IF eError <> MotionlinxAI_Error_States.NO_ERROR  OR eError = MotionlinxAI_Error_States.MOTOR_UNDERVOLTAGE  THEN
	IF (bMotorDisconnected AND NOT bMotorExpected)  THEN
		_Error := FALSE;
	ELSE
		_Error := TRUE;
		eError := eError;
	
			
//		IF oClearMotorError = 0 THEN
//			oClearMotorError := 1;
//		ELSIF oClearMotorError = 1 THEN
//			oClearMotorError := 0;
//		END_IF;
	END_IF

ELSE
	_Error := FALSE;
END_IF;
END_ACTION

PROPERTY HasFault : BOOL
GET
HasFault := eMotionlinxAIState < MotionlinxAI_States.HOMING;// or bCommunicationsFailed;
END_GET
END_PROPERTY

METHOD PROTECTED HMICommunication
VAR_INPUT
END_VAR
SUPER^.HMICommunication();

//Handle the requests to extend and retract
IF ComponentBase_HMI.Status.HMIControlAvailable THEN
	IF MotionlinxAI_HMI.Command.Extend THEN
//		Extend();
	ELSIF MotionlinxAI_HMI.Command.Retract THEN
//		Retract();
	END_IF
END_IF

//Update HMI status info
//Cylinder_HMI.Status.Extended	:= _Extended;
//Cylinder_HMI.Status.Extending	:= _Extending;
//Cylinder_HMI.Status.Retracted	:= _Retracted;
//Cylinder_HMI.Status.Retracting	:= _Retracting;
//Cylinder_HMI.Config.ExtendTime	:= _ExtendTime;
//Cylinder_HMI.Config.RetractTime := _RetractTime;
END_METHOD

//! @summary Basic component initialization logic
METHOD PROTECTED Initialize : BOOL;

//! @description This method is called by <c>CyclicLogic()</c> as required



//Set the cylinder to retracted
//oMotorAccel	:= 500;		//From recipe value here
//IF Output THEN
//	_Extended  := TRUE;
//	_Retracted := FALSE;
//ELSE
//	_Extended  := FALSE;
//	_Retracted := TRUE;
//END_IF



//Call base class Initialize
Initialize := SUPER^.Initialize();
END_METHOD

PROPERTY IsReady : BOOL
GET
IsReady := eMotionlinxAIState > MotionlinxAI_States.HOMING;
END_GET
END_PROPERTY

PROPERTY MaxSpeed : uint
SET
uMaxSpeed	:= MaxSpeed;
END_SET
END_PROPERTY

METHOD PROTECTED Monitoring
VAR_INPUT
END_VAR
_Busy	 := NOT Stopped;//MotionlinxAI_Motor_Status:=3 OR MotionlinxAI_Motor_Status:=4 ;
_Error	 := eError>0 OR eMotionlinxAIState < MotionlinxAI_States.HOMING;;
_ErrorID := eError;
SUPER^.Monitoring();
END_METHOD

PROPERTY MotorDisconnected : bool
GET
MotorDisconnected	:= bMotorDisconnected;
END_GET
END_PROPERTY

METHOD RaiseAlarm2Args
VAR_IN_OUT
	Alarm : FB_TcAlarm; //Alarm to be raised
END_VAR

VAR_INPUT
	String_1 : STRING; //First String Parameter (The Name of this component will be applied first automatically)
	String_2 : STRING; //Second String Parameter
END_VAR
F_RaiseAlarmWithStringParameters(Alarm	  := Alarm,
								 String_1 := Name,
								 String_2 := String_1,
								 String_3 := String_2);
END_METHOD

METHOD Start : BOOL
VAR_INPUT
END_VAR
IF bEnabled THEN 
	oMotorControl.0 := TRUE;
	oMotorBrakeMode  := 2;
END_IF
END_METHOD

METHOD Stop
VAR_INPUT
END_VAR
oMotorControl.0 := FALSE;
oMotorBrakeMode := 2;
END_METHOD

PROPERTY Stopped : bool
GET
Stopped	:= bAxis_Stopped;
END_GET
END_PROPERTY

PROPERTY Velocity : int
SET
nRequestedSpeed	:= Velocity;
//Recipe.Axis.Acceleration := Acceleration;
END_SET
END_PROPERTY

END_FUNCTION_BLOCK

// ---- Machine/Components/MotionLinxAI/Controller/FB_MotionlinxAI_Controller.TcPOU
(*	
*)
FUNCTION_BLOCK FB_MotionlinxAI_Controller EXTENDS FB_ComponentBase IMPLEMENTS I_MotionlinxAI_Controller_Sts
VAR
//Inputs
	iSensors AT%I* : INT;
	iSysDiagnostics AT%I* : BYTE;
//	Drive_1_Left	  : FB_MotionlinxAI_Axis (Main_Sensor	:= iSensors.4, Aux_Sensor	:= iSensors.0 ):= (Name := 'Left Drive 1');
//	Drive_2_Right	  : FB_MotionlinxAI_Axis (Main_Sensor	:= iSensors.6, Aux_Sensor	:= iSensors.2 ):= (Name := 'Right Drive 2');
	

	//Output
	oServoControl AT%Q* : INT;
	oSetPin2Out AT%Q* : BYTE;
	oClearMotorError  AT%Q* : BYTE;
	
	//From Other project, can possibly be modifdied a bit
	//Connection Monitoring//
	bWCState AT%I* : BOOL; //0 is Data Valid, 1 is Data Invalid
	
	tonCommunicationsFailed : TON;
	bCommunicationsFailed : BOOL;
	
	bInputToggle AT%I* : BOOL;

	// Internal variables
	//Error Resetting//
	bError : BOOL;
	tpErrorReset : TP;
	
	//Speed Limits//
	rPGDMaxSpeed : REAL := 536.0;
	rPGDMinSpeed : REAL := 3888.0;
	
	
	//Motor Status//
	eMotorStatus: MotionlinxAI_Motor_Status;
	eErrorRecord : MotionlinxAI_Error_States;
	_stController_Sts	:ST_Controller_Status;

	
	
	
//	_ExtendRequest	: BOOL;
//	_RetractRequest : BOOL;
//	_Extended		: BOOL;
//	_Retracted		: BOOL;
//	_Extending		: BOOL;
//	_Retracting		: BOOL;
//	_ExtendTime		: LREAL := 1000; // Default time 1s
//	_RetractTime	: LREAL := 1000; // Default time 1s

//	// Timer for Extend/Retract
//	Extend_TON	  : TON;
//	Retract_TON	  : TON;
//	Extend_RTRIG  : R_TRIG;
//	Retract_RTRIG : R_TRIG;

	//HMI 
	MotionlinxAI_Controller_HMI : ST_MotionlinxAI_Axis_HMI;
END_VAR

PROPERTY CommunicationsFailed : bool
GET
CommunicationsFailed	:= bCommunicationsFailed;
END_GET
END_PROPERTY

PROPERTY Controller_Status : ST_Controller_Status
GET
Controller_Status	:= _stController_Sts;
END_GET
END_PROPERTY

METHOD PROTECTED CreateEvents
VAR_INPUT
END_VAR
SUPER^.CreateEvents();
END_METHOD

METHOD CyclicLogic
VAR

END_VAR
//////////Error Handling//////////
errorCheck();
_stController_Sts.Sensors	:= iSensors;
_stController_Sts.bEnabled	:= isEnabled;
_stController_Sts.HasFault	:= HasFault;

//////////Set Speed Limits//////////
//uLMinSpeed := 15+uLMaxSpeed/100;
//uRMinSpeed := 15+uRMaxSpeed/100;
//////////Set Speeds//////////
//oMotorLSpeed := LIMIT(UINT_TO_INT(uLMinSpeed),UINT_TO_INT(nRequestedSpeedLeft),UINT_TO_INT(uLMaxSpeed));
//oMotorRSpeed := LIMIT(UINT_TO_INT(uRMinSpeed),UINT_TO_INT(nRequestedSpeedRight),UINT_TO_INT(uRMaxSpeed));


////////////Stop On Disable//////////
//IF NOT bEnabled THEN
//	oMotorLDecel := oMotorRDecel := 500;	
//	oMotorLControl.0 := oMotorRControl.0 := FALSE;
//ELSE
//	oMotorLDecel := oMotorRDecel := 500;
//END_IF;



//////////Communications Monitoring//////////
tonCommunicationsFailed(IN:= bWCState, PT:= T#10S, Q => bCommunicationsFailed);


//One shot the requests


//Handle Extend
//IF Extend_RTRIG.Q THEN
//	Output			:= TRUE;
//	_Extending		:= TRUE;
//	_Retracting		:= FALSE;
//	_Retracted		:= FALSE;
//	_RetractRequest := FALSE;
//END_IF

//Handle Retract
//IF Retract_RTRIG.Q THEN
//	Output		   := FALSE;
//	_Extending	   := FALSE;
//	_Retracting	   := TRUE;
//	_Extended	   := FALSE;
//	_ExtendRequest := FALSE;
//END_IF

//Handle the time to Extend/Retract
//Extend_TON(IN := _Extending, PT := LREAL_TO_TIME(_ExtendTime));
//Retract_TON(IN := _Retracting, PT := LREAL_TO_TIME(_RetractTime));
//IF Extend_TON.Q THEN
//	_Extended  := TRUE;
//	_Extending := FALSE;
//END_IF

//IF Retract_TON.Q THEN
//	_Retracted	:= TRUE;
//	_Retracting := FALSE;
//END_IF

SUPER^.CyclicLogic();
END_METHOD

METHOD Disable : BOOL
(*BRAKING MODES:
	0 : NORMAL - HOLDS IN PLACE BY SHORTING WINDINGS
	1 : FREE - NOT HELD IN PLACE
	2 : SERVO - MAINTAINS POSITION BASED ON HALLS EFFECT SENSOR*)
//oMotorLDecel := oMotorRDecel := 500;
//bEnabled := FALSE;
//(*oMotorLControl.0 := FALSE;
//oMotorRControl.0 := FALSE;*)
//oMotorLBrakeMode := oMotorRBrakeMode := 2;
END_METHOD

METHOD EmergencyStop : BOOL
(*BRAKING MODES:
	0 : NORMAL - HOLDS IN PLACE BY SHORTING WINDINGS
	1 : FREE - NOT HELD IN PLACE
	2 : SERVO - MAINTAINS POSITION BASED ON HALLS EFFECT SENSOR*)
//oMotorLDecel := oMotorRDecel := 1;
//bEnabled := FALSE;
//(*oMotorLControl.0 := FALSE;
//oMotorRControl.0 := FALSE;*)
//oMotorLBrakeMode := oMotorRBrakeMode := 0;
END_METHOD

METHOD Enable : BOOL
(*BRAKING MODES:
	0 : NORMAL - HOLDS IN PLACE BY SHORTING WINDINGS
	1 : FREE - NOT HELD IN PLACE
	2 : SERVO - MAINTAINS POSITION BASED ON HALLS EFFECT SENSOR*)
//bEnabled := TRUE;
//oMotorLBrakeMode := oMotorRBrakeMode := 2;
END_METHOD

ACTION errorCheck:
//oClearMotorError := 0;




//IF eErrorLeft <> MotionlinxAI_Error_States.NO_ERROR OR eErrorRight <> MotionlinxAI_Error_States.NO_ERROR OR eErrorLeft = MotionlinxAI_Error_States.MOTOR_UNDERVOLTAGE OR eErrorRight = MotionlinxAI_Error_States.MOTOR_UNDERVOLTAGE THEN
//	IF (bLeftMotorDisconnected AND NOT bLeftMotorExpected) OR (bRightMotorDisconnected AND NOT bRightMotorExpected) THEN
//		bError := FALSE;
//	ELSE
//		bError := TRUE;
//	//	eErrorRecordLeft := eErrorLeft;
//	//	eErrorRecordRight := eErrorRight;
			
//		IF oClearMotorError = 0 THEN
//			oClearMotorError := 1;
//		ELSIF oClearMotorError = 1 THEN
//			oClearMotorError := 0;
//		END_IF;
//	END_IF

//ELSE
//	bError := FALSE;
//END_IF;
END_ACTION

PROPERTY FaultLocation : STRING(50)
GET
//FaultLocation := sDriveName;
END_GET
END_PROPERTY

PROPERTY HasFault : BOOL
GET
//HasFault := eMotionlinxAIState < MotionlinxAI_States.HOMING or bCommunicationsFailed;
END_GET
END_PROPERTY

METHOD PROTECTED HMICommunication
VAR_INPUT
END_VAR
SUPER^.HMICommunication();

//Handle the requests to extend and retract
IF ComponentBase_HMI.Status.HMIControlAvailable THEN
	IF MotionlinxAI_Controller_HMI.Command.Extend THEN
	//	Extend();
	ELSIF MotionlinxAI_Controller_HMI.Command.Retract THEN
	//	Retract();
	END_IF
END_IF

//Update HMI status info
//MotionlinxAI_Controller_HMI.Status.Extended	:= _Extended;
//MotionlinxAI_Controller_HMI.Status.Extending	:= _Extending;
//MotionlinxAI_Controller_HMI.Status.Retracted	:= _Retracted;
//MotionlinxAI_Controller_HMI.Status.Retracting	:= _Retracting;
//MotionlinxAI_Controller_HMI.Config.ExtendTime	:= _ExtendTime;
//MotionlinxAI_Controller_HMI.Config.RetractTime := _RetractTime;
END_METHOD

//! @summary Basic component initialization logic
METHOD PROTECTED Initialize : BOOL;

//! @description This method is called by <c>CyclicLogic()</c> as required
//Set the cylinder to retracted
//IF Output THEN
//	_Extended  := TRUE;
//	_Retracted := FALSE;
//ELSE
//	_Extended  := FALSE;
//	_Retracted := TRUE;
//END_IF

//_Extending		:= FALSE;
//_ExtendRequest	:= FALSE;
//_Retracting		:= FALSE;
//_RetractRequest := FALSE;

//Call base class Initialize
Initialize := SUPER^.Initialize();
END_METHOD

PROPERTY IsEnabled : BOOL
GET
//IsEnabled := bEnabled;
END_GET
END_PROPERTY

PROPERTY IsReady : BOOL
GET
//IsReady := eMotionlinxAIState > MotionlinxAI_States.HOMING;
END_GET
END_PROPERTY

METHOD PROTECTED Monitoring
VAR_INPUT
END_VAR
//_Busy	 := _Extending OR _Retracting;
_Error	 := bCommunicationsFailed;
_ErrorID := 0;
SUPER^.Monitoring();
END_METHOD

PROPERTY Sensors : int
GET
Sensors	:= iSensors;
END_GET
END_PROPERTY

ACTION stop:
//oMotorLControl.0 := FALSE;
//oMotorRControl.0 := FALSE;
END_ACTION

END_FUNCTION_BLOCK

// ---- Machine/Components/Robots/UR/fbUR.TcPOU
FUNCTION_BLOCK fbUR
VAR_INPUT
END_VAR
VAR_OUTPUT
END_VAR
VAR	
	EIO_UR_Outputs AT %Q* : UR_Output_Data;
	EIO_UR_Inputs  AT %I* : UR_Safety_Bits_Data;

	bBrakeRelease AT %Q* : BOOL;
	
	rtRobotSafe			: R_TRIG;
	
	tpBrakeRelease		: TP;
	
	tonPowerUpRobot		: TON;
	tpPowerOnPulse		: TP;
END_VAR

rtRobotSafe(CLK := EIO_UR_Inputs.data.ibNormalMode OR EIO_UR_Inputs.data.ibReducedMode);
EIO_UR_Outputs.data.obBrakeRelease := bBrakeRelease;

tpBrakeRelease(IN := GVL_Safety.PALLETISER_ESTOP_OK AND NOT (GVL_HMI.ibResetButton OR GVL_HMI.bHMIResetButton), PT := T#1S, Q => bBrakeRelease);

tonPowerUpRobot(IN:= NOT GVL_Palletiser.ibURPowered, PT := T#20S);
tpPowerOnPulse(IN := tonPowerUpRobot.Q, Q => GVL_Palletiser.obURPowerOn, PT := T#0.5S);

END_FUNCTION_BLOCK

// ---- Machine/Components/Contactor/FB_Contactor.TcPOU
(*	This FB is used for a single output solenoid 
	It uses the times to say when Extended/Retracted  	
	It starts assuming retracted and the output off.
*)
FUNCTION_BLOCK FB_Contactor EXTENDS FB_ComponentBase IMPLEMENTS I_Contactor
VAR
    //Output
    Output AT %Q* : BOOL;

    // Internal variables
    _ExtendRequest  : BOOL;
    _RetractRequest : BOOL;
    _Extended       : BOOL;
    _Retracted      : BOOL;
    _Extending      : BOOL;
    _Retracting     : BOOL;
    _ExtendTime     : LREAL := 1000; // Default time 1s
    _RetractTime    : LREAL := 1000; // Default time 1s

    // Timer for Extend/Retract
    Extend_TON    : TON;
    Retract_TON   : TON;
    Extend_RTRIG  : R_TRIG;
    Retract_RTRIG : R_TRIG;

    //HMI 
    Contactor_HMI : ST_Contactor_HMI;
END_VAR

METHOD PROTECTED CreateEvents
VAR_INPUT
END_VAR
SUPER^.CreateEvents();
END_METHOD

METHOD CyclicLogic
//One shot the requests
Extend_RTRIG(CLK := _ExtendRequest);
Retract_RTRIG(CLK := _RetractRequest);

//Handle Extend
IF Extend_RTRIG.Q THEN
    Output          := TRUE;
    _Extending      := TRUE;
    _Retracting     := FALSE;
    _Retracted      := FALSE;
    _RetractRequest := FALSE;
END_IF

//Handle Retract
IF Retract_RTRIG.Q THEN
    Output         := FALSE;
    _Extending     := FALSE;
    _Retracting    := TRUE;
    _Extended      := FALSE;
    _ExtendRequest := FALSE;
END_IF

//Handle the time to Extend/Retract
Extend_TON(IN := _Extending, PT := LREAL_TO_TIME(_ExtendTime));
Retract_TON(IN := _Retracting, PT := LREAL_TO_TIME(_RetractTime));
IF Extend_TON.Q THEN
    _Extended  := TRUE;
    _Extending := FALSE;
END_IF

IF Retract_TON.Q THEN
    _Retracted  := TRUE;
    _Retracting := FALSE;
END_IF

SUPER^.CyclicLogic();
END_METHOD

METHOD Extend
_ExtendRequest  := TRUE;
_RetractRequest := FALSE;
END_METHOD

PROPERTY Extended : BOOL
GET
Extended := _Extended;
END_GET
END_PROPERTY

PROPERTY ExtendTime : LREAL
GET
ExtendTime := _ExtendTime;
END_GET
SET
END_SET
END_PROPERTY

METHOD PROTECTED HMICommunication
VAR_INPUT
END_VAR
SUPER^.HMICommunication();

//Handle the requests to extend and retract
IF ComponentBase_HMI.Status.HMIControlAvailable THEN
    IF Contactor_HMI.Command.Extend THEN
        Extend();
    ELSIF Contactor_HMI.Command.Retract THEN
        Retract();
    END_IF
END_IF

//Update HMI status info
Contactor_HMI.Status.Extended    := _Extended;
Contactor_HMI.Status.Extending   := _Extending;
Contactor_HMI.Status.Retracted   := _Retracted;
Contactor_HMI.Status.Retracting  := _Retracting;
Contactor_HMI.Config.ExtendTime  := _ExtendTime;
Contactor_HMI.Config.RetractTime := _RetractTime;
END_METHOD

//! @summary Basic component initialization logic
METHOD PROTECTED Initialize : BOOL;

//! @description This method is called by <c>CyclicLogic()</c> as required
//Set the Contactor to retracted
IF Output THEN
    _Extended  := TRUE;
    _Retracted := FALSE;
ELSE
    _Extended  := FALSE;
    _Retracted := TRUE;
END_IF

_Extending      := FALSE;
_ExtendRequest  := FALSE;
_Retracting     := FALSE;
_RetractRequest := FALSE;

//Call base class Initialize
Initialize := SUPER^.Initialize();
END_METHOD

METHOD PROTECTED Monitoring
VAR_INPUT
END_VAR
_Busy    := _Extending OR _Retracting;
_Error   := FALSE;
_ErrorID := 0;
SUPER^.Monitoring();
END_METHOD

METHOD Retract
_ExtendRequest  := FALSE;
_RetractRequest := TRUE;
END_METHOD

PROPERTY Retracted : BOOL
GET
Retracted := _Retracted;
END_GET
END_PROPERTY

PROPERTY RetractTime : LREAL
GET
RetractTime := _RetractTime;
END_GET
SET
_RetractTime := RetractTime;
END_SET
END_PROPERTY

END_FUNCTION_BLOCK

// ---- Machine/Components/Contactor/FB_Contactor_Dual_InOut.TcPOU
(*	This FB is used for a single output solenoid 
	It uses the single input to say when Extended  	
	It starts assuming retracted and the output off.
*)
FUNCTION_BLOCK FB_Contactor_Dual_InOut EXTENDS FB_ComponentBase IMPLEMENTS I_Contactor
VAR
    //Output
    qExtend 				AT %Q* : BOOL;
	qRetract				AT %Q* : BOOL;
//	FeedBackExtended	AT %I* : BOOL;	//This could be an sensor FB
//	FeedBackRetracted	AT %I* : BOOL;	//This could be an sensor FB
	ExtendedSensor		:FB_DigitalSensor		:= (Name := 'Sensor', DebounceMode := E_DebounceMode.SimpleFlickerFilter, DebounceTime := T#250MS, Inverted    := FALSE, SimulationInput:= FALSE, SimulationMode := E_SensorSimulationMode.InputDriven) ;	//I_DigitalSensorBase;
	RetractedSensor		:FB_DigitalSensor		:= (Name := 'Sensor', DebounceMode := E_DebounceMode.SimpleFlickerFilter, DebounceTime := T#250MS, Inverted    := FALSE, SimulationInput:= FALSE, SimulationMode := E_SensorSimulationMode.InputDriven) ;

	
	 // List of Components
 //   ipComponents_Init :
  //     ARRAY[1..Parameters_PackML_Base.MAX_NO_OF_COMPONENTS] OF I_ComponentBase := [ ExtendedSensor];

    // Internal variables
    _ExtendRequest  : BOOL;
    _RetractRequest : BOOL;
    _Extended       : BOOL;
    _Retracted      : BOOL;
    _Extending      : BOOL;
    _Retracting     : BOOL;
    _ExtendTime     : LREAL := 1000; // Default time 1s
    _RetractTime    : LREAL := 1000; // Default time 1s

    // Timer for Extend/Retract
    Extend_TON    : TON;
    Retract_TON   : TON;
    Extend_RTRIG  : R_TRIG;
	ExtendIN_RTRIG: R_TRIG;
    Retract_RTRIG : R_TRIG;
	RetractIN_RTRIG : R_TRIG;

    //HMI 
    Contactor_HMI : ST_Contactor_HMI;
END_VAR

METHOD PROTECTED CreateEvents
VAR_INPUT
END_VAR
SUPER^.CreateEvents();
END_METHOD

METHOD CyclicLogic
//IO
ExtendedSensor();
RetractedSensor();

//One shot the requests
Extend_RTRIG(CLK := _ExtendRequest);
Retract_RTRIG(CLK := _RetractRequest);

//Handle Extend
IF Extend_RTRIG.Q THEN
    qEXTEND          := TRUE;
	qRETRACT			:= FALSE;
    _Extending      := TRUE;
    _Retracting     := FALSE;
    _Retracted      := FALSE;
    _RetractRequest := FALSE;
END_IF

//Handle Retract
IF Retract_RTRIG.Q THEN
    qEXTEND          := FALSE;
	qRETRACT			:= TRUE;
    _Extending     := FALSE;
    _Retracting    := TRUE;
    _Extended      := FALSE;
    _ExtendRequest := FALSE;
END_IF

//Handle the triggers to Extend/Retract
ExtendIN_RTRIG	(clk:=ExtendedSensor.Active); 
RetractIN_RTRIG	(clk:= RetractedSensor.Active);
//Extend_TON(IN := _Extending, PT := LREAL_TO_TIME(_ExtendTime));
//Retract_TON(IN := _Retracting, PT := LREAL_TO_TIME(_RetractTime));
IF ExtendIN_RTRIG.Q THEN
    _Extended  := TRUE;
    _Extending := FALSE;
END_IF

IF RetractIN_RTRIG.Q THEN
    _Retracted  := TRUE;
    _Retracting := FALSE;
END_IF

SUPER^.CyclicLogic();
END_METHOD

METHOD Extend
_ExtendRequest  := TRUE;
_RetractRequest := FALSE;
END_METHOD

PROPERTY Extended : BOOL
GET
Extended := _Extended;
END_GET
END_PROPERTY

PROPERTY ExtendTime : LREAL
GET
ExtendTime := _ExtendTime;
END_GET
SET
END_SET
END_PROPERTY

METHOD PROTECTED HMICommunication
VAR_INPUT
END_VAR
SUPER^.HMICommunication();

//Handle the requests to extend and retract
IF ComponentBase_HMI.Status.HMIControlAvailable THEN
    IF Contactor_HMI.Command.Extend THEN
        Extend();
    ELSIF Contactor_HMI.Command.Retract THEN
        Retract();
    END_IF
END_IF

//Update HMI status info
Contactor_HMI.Status.Extended    := _Extended;
Contactor_HMI.Status.Extending   := _Extending;
Contactor_HMI.Status.Retracted   := _Retracted;
Contactor_HMI.Status.Retracting  := _Retracting;
Contactor_HMI.Config.ExtendTime  := _ExtendTime;
Contactor_HMI.Config.RetractTime := _RetractTime;
END_METHOD

//! @summary Basic component initialization logic
METHOD PROTECTED Initialize : BOOL;

//! @description This method is called by <c>CyclicLogic()</c> as required
//Set the Contactor to retracted
IF Extended THEN
    _Extended  := TRUE;
    _Retracted := FALSE;
ELSIF retracted THEN
    _Extended  := FALSE;
    _Retracted := TRUE;
END_IF

_Extending      := FALSE;
_ExtendRequest  := FALSE;
_Retracting     := FALSE;
_RetractRequest := FALSE;

//Call base class Initialize
Initialize := SUPER^.Initialize();
END_METHOD

METHOD PROTECTED Monitoring
VAR_INPUT
END_VAR
_Busy    := _Extending OR _Retracting;
_Error   := FALSE;
_ErrorID := 0;
SUPER^.Monitoring();
END_METHOD

METHOD Retract
_ExtendRequest  := FALSE;
_RetractRequest := TRUE;
END_METHOD

PROPERTY Retracted : BOOL
GET
Retracted := _Retracted;
END_GET
END_PROPERTY

PROPERTY RetractTime : LREAL
GET
RetractTime := _RetractTime;
END_GET
SET
_RetractTime := RetractTime;
END_SET
END_PROPERTY

END_FUNCTION_BLOCK

// ---- Machine/Components/Contactor/FB_Contactor_With_Dual_Feedback.TcPOU
(*	This FB is used for a single output solenoid 
	It uses the single input to say when Extended  	
	It starts assuming retracted and the output off.
*)
FUNCTION_BLOCK FB_Contactor_With_Dual_Feedback EXTENDS FB_ComponentBase IMPLEMENTS I_Contactor
VAR
    //Output
    Output 				AT %Q* : BOOL;
//	FeedBackExtended	AT %I* : BOOL;	//This could be an sensor FB
//	FeedBackRetracted	AT %I* : BOOL;	//This could be an sensor FB
	ExtendedSensor		:FB_DigitalSensor		:= (Name := 'Sensor', DebounceMode := E_DebounceMode.SimpleFlickerFilter, DebounceTime := T#250MS, Inverted    := FALSE, SimulationInput:= FALSE, SimulationMode := E_SensorSimulationMode.InputDriven) ;		//I_DigitalSensorBase;
	RetractedSensor		:FB_DigitalSensor		:= (Name := 'Sensor', DebounceMode := E_DebounceMode.SimpleFlickerFilter, DebounceTime := T#250MS, Inverted    := FALSE, SimulationInput:= FALSE, SimulationMode := E_SensorSimulationMode.InputDriven) ;

	
	 // List of Components
 //   ipComponents_Init :
  //     ARRAY[1..Parameters_PackML_Base.MAX_NO_OF_COMPONENTS] OF I_ComponentBase := [ ExtendedSensor];

    // Internal variables
    _ExtendRequest  : BOOL;
    _RetractRequest : BOOL;
    _Extended       : BOOL;
    _Retracted      : BOOL;
    _Extending      : BOOL;
    _Retracting     : BOOL;
    _ExtendTime     : LREAL := 1000; // Default time 1s
    _RetractTime    : LREAL := 1000; // Default time 1s

    // Timer for Extend/Retract
    Extend_TON    : TON;
    Retract_TON   : TON;
    Extend_RTRIG  : R_TRIG;
    Retract_RTRIG : R_TRIG;

    //HMI 
    Contactor_HMI : ST_Contactor_HMI;
END_VAR

METHOD PROTECTED CreateEvents
VAR_INPUT
END_VAR
SUPER^.CreateEvents();
END_METHOD

METHOD CyclicLogic
//IO
ExtendedSensor();
RetractedSensor();

//One shot the requests
Extend_RTRIG(CLK := _ExtendRequest);
Retract_RTRIG(CLK := _RetractRequest);

//Handle Extend
IF Extend_RTRIG.Q THEN
    Output          := TRUE;
    _Extending      := TRUE;
    _Retracting     := FALSE;
    _Retracted      := FALSE;
    _RetractRequest := FALSE;
END_IF

//Handle Retract
IF Retract_RTRIG.Q THEN
    Output         := FALSE;
    _Extending     := FALSE;
    _Retracting    := TRUE;
    _Extended      := FALSE;
    _ExtendRequest := FALSE;
END_IF

//Handle the time to Extend/Retract
Extend_TON(IN := _Extending, PT := LREAL_TO_TIME(_ExtendTime));
Retract_TON(IN := _Retracting, PT := LREAL_TO_TIME(_RetractTime));
IF ExtendedSensor.Active THEN
    _Extended  := TRUE;
    _Extending := FALSE;
END_IF

IF RetractedSensor.Active THEN
    _Retracted  := TRUE;
    _Retracting := FALSE;
END_IF

SUPER^.CyclicLogic();
END_METHOD

METHOD Extend
_ExtendRequest  := TRUE;
_RetractRequest := FALSE;
END_METHOD

PROPERTY Extended : BOOL
GET
Extended := _Extended;
END_GET
END_PROPERTY

PROPERTY ExtendTime : LREAL
GET
ExtendTime := _ExtendTime;
END_GET
SET
END_SET
END_PROPERTY

METHOD PROTECTED HMICommunication
VAR_INPUT
END_VAR
SUPER^.HMICommunication();

//Handle the requests to extend and retract
IF ComponentBase_HMI.Status.HMIControlAvailable THEN
    IF Contactor_HMI.Command.Extend THEN
        Extend();
    ELSIF Contactor_HMI.Command.Retract THEN
        Retract();
    END_IF
END_IF

//Update HMI status info
Contactor_HMI.Status.Extended    := _Extended;
Contactor_HMI.Status.Extending   := _Extending;
Contactor_HMI.Status.Retracted   := _Retracted;
Contactor_HMI.Status.Retracting  := _Retracting;
Contactor_HMI.Config.ExtendTime  := _ExtendTime;
Contactor_HMI.Config.RetractTime := _RetractTime;
END_METHOD

//! @summary Basic component initialization logic
METHOD PROTECTED Initialize : BOOL;

//! @description This method is called by <c>CyclicLogic()</c> as required
//Set the Contactor to retracted
IF Output THEN
    _Extended  := TRUE;
    _Retracted := FALSE;
ELSE
    _Extended  := FALSE;
    _Retracted := TRUE;
END_IF

_Extending      := FALSE;
_ExtendRequest  := FALSE;
_Retracting     := FALSE;
_RetractRequest := FALSE;

//Call base class Initialize
Initialize := SUPER^.Initialize();
END_METHOD

METHOD PROTECTED Monitoring
VAR_INPUT
END_VAR
_Busy    := _Extending OR _Retracting;
_Error   := FALSE;
_ErrorID := 0;
SUPER^.Monitoring();
END_METHOD

METHOD Retract
_ExtendRequest  := FALSE;
_RetractRequest := TRUE;
END_METHOD

PROPERTY Retracted : BOOL
GET
Retracted := _Retracted;
END_GET
END_PROPERTY

PROPERTY RetractTime : LREAL
GET
RetractTime := _RetractTime;
END_GET
SET
_RetractTime := RetractTime;
END_SET
END_PROPERTY

END_FUNCTION_BLOCK

// ---- Machine/Components/Contactor/FB_Contactor_With_Single_Feedback.TcPOU
(*	This FB is used for a single output solenoid 
	It uses the single input to say when Extended  	
	It starts assuming retracted and the output off.
*)
FUNCTION_BLOCK FB_Contactor_With_Single_Feedback EXTENDS FB_ComponentBase IMPLEMENTS I_Contactor
VAR
    //Output
    Output 				AT %Q* : BOOL;
//	FeedBackExtended	AT %I* : BOOL;	//This could be an sensor FB
	ExtendedSensor		:FB_DigitalSensor		:= (Name := 'Sensor', DebounceMode := E_DebounceMode.SimpleFlickerFilter, DebounceTime := T#250MS, Inverted    := FALSE, SimulationInput:= FALSE, SimulationMode := E_SensorSimulationMode.InputDriven) ;

    // Internal variables
    _ExtendRequest  : BOOL;
    _RetractRequest : BOOL;
    _Extended       : BOOL;
    _Retracted      : BOOL;
    _Extending      : BOOL;
    _Retracting     : BOOL;
    _ExtendTime     : LREAL := 1000; // Default time 1s
    _RetractTime    : LREAL := 1000; // Default time 1s

    // Timer for Extend/Retract
    Extend_TON    : TON;
    Retract_TON   : TON;
    Extend_RTRIG  : R_TRIG;
    Retract_RTRIG : R_TRIG;

    //HMI 
    Contactor_HMI : ST_Contactor_HMI;
END_VAR

METHOD PROTECTED CreateEvents
VAR_INPUT
END_VAR
SUPER^.CreateEvents();
END_METHOD

METHOD CyclicLogic
//One shot the requests
Extend_RTRIG(CLK := _ExtendRequest);
Retract_RTRIG(CLK := _RetractRequest);

//Handle Extend
IF Extend_RTRIG.Q THEN
    Output          := TRUE;
    _Extending      := TRUE;
    _Retracting     := FALSE;
    _Retracted      := FALSE;
    _RetractRequest := FALSE;
END_IF

//Handle Retract
IF Retract_RTRIG.Q THEN
    Output         := FALSE;
    _Extending     := FALSE;
    _Retracting    := TRUE;
    _Extended      := FALSE;
    _ExtendRequest := FALSE;
END_IF

//Handle the time to Extend/Retract
Extend_TON(IN := _Extending, PT := LREAL_TO_TIME(_ExtendTime));
Retract_TON(IN := _Retracting, PT := LREAL_TO_TIME(_RetractTime));
IF ExtendedSensor.Active THEN
    _Extended  := TRUE;
    _Extending := FALSE;
END_IF

IF Retract_TON.Q AND NOT ExtendedSensor.Active THEN
    _Retracted  := TRUE;
    _Retracting := FALSE;
END_IF

SUPER^.CyclicLogic();
END_METHOD

METHOD Extend
_ExtendRequest  := TRUE;
_RetractRequest := FALSE;
END_METHOD

PROPERTY Extended : BOOL
GET
Extended := _Extended;
END_GET
END_PROPERTY

PROPERTY ExtendTime : LREAL
GET
ExtendTime := _ExtendTime;
END_GET
SET
END_SET
END_PROPERTY

METHOD PROTECTED HMICommunication
VAR_INPUT
END_VAR
SUPER^.HMICommunication();

//Handle the requests to extend and retract
IF ComponentBase_HMI.Status.HMIControlAvailable THEN
    IF Contactor_HMI.Command.Extend THEN
        Extend();
    ELSIF Contactor_HMI.Command.Retract THEN
        Retract();
    END_IF
END_IF

//Update HMI status info
Contactor_HMI.Status.Extended    := _Extended;
Contactor_HMI.Status.Extending   := _Extending;
Contactor_HMI.Status.Retracted   := _Retracted;
Contactor_HMI.Status.Retracting  := _Retracting;
Contactor_HMI.Config.ExtendTime  := _ExtendTime;
Contactor_HMI.Config.RetractTime := _RetractTime;
END_METHOD

//! @summary Basic component initialization logic
METHOD PROTECTED Initialize : BOOL;

//! @description This method is called by <c>CyclicLogic()</c> as required
//Set the Contactor to retracted
IF Output THEN
    _Extended  := TRUE;
    _Retracted := FALSE;
ELSE
    _Extended  := FALSE;
    _Retracted := TRUE;
END_IF

_Extending      := FALSE;
_ExtendRequest  := FALSE;
_Retracting     := FALSE;
_RetractRequest := FALSE;

//Call base class Initialize
Initialize := SUPER^.Initialize();
END_METHOD

METHOD PROTECTED Monitoring
VAR_INPUT
END_VAR
_Busy    := _Extending OR _Retracting;
_Error   := FALSE;
_ErrorID := 0;
SUPER^.Monitoring();
END_METHOD

METHOD Retract
_ExtendRequest  := FALSE;
_RetractRequest := TRUE;
END_METHOD

PROPERTY Retracted : BOOL
GET
Retracted := _Retracted;
END_GET
END_PROPERTY

PROPERTY RetractTime : LREAL
GET
RetractTime := _RetractTime;
END_GET
SET
_RetractTime := RetractTime;
END_SET
END_PROPERTY

END_FUNCTION_BLOCK

// ---- Machine/Components/Drives/Omron/FB_Omron_Inv.TcPOU
FUNCTION_BLOCK FB_Omron_Inv EXTENDS FB_ComponentBase IMPLEMENTS iDM_DriveHealth
VAR
	// Data
	_SetTemperature	   : LREAL;
	_ActualTemperature : LREAL;

	// IO
	_Heat AT %Q* : BOOL;

	// Other items
	RequestedState : eDriveStates	:= eDriveStates.AWAITING_RESET;	
	DriveState : eDriveStates 		:= eDriveStates.FAULT;

	bEnabled : BOOL;
	bInitReversed : BOOL;
	bError : BOOL;
	
	
	eDeviceStatus : eOmronStatus;
	
	bRunningForward : BOOL;
	bRunningReverse : BOOL;
	bFault : BOOL;
	bWarning : BOOL;
	bRemoteEnabled : BOOL;
	bFrequencyMatching : BOOL;
	bConnectionError : BOOL;
	bECDisconnected : BOOL;
	
	blinkErrorAck : FB_BLINKER_PLAY;
	
	tpErrorReset : TP;
	bResetReq : BOOL;
	
	sDriveName : STRING(50);
	tonFailedStartTimeout : TON;
	bResetTried: BOOL;
	
	
//	TempUpdate	 : TON;
//	_InTempRange : BOOL;
END_VAR

ACTION aInputMapping:
bDI1 := stDeviceMapping.inInputTerminal.2;
bDI2 := stDeviceMapping.inInputTerminal.3;
bDI3 := stDeviceMapping.inInputTerminal.4;
bDI4 := stDeviceMapping.inInputTerminal.5;
bDI5 := stDeviceMapping.inInputTerminal.6;
bDI6 := stDeviceMapping.inInputTerminal.0; 
bDI7 := stDeviceMapping.inInputTerminal.1;
bEN1 := stDeviceMapping.inInputTerminal.11;
bEN2 := stDeviceMapping.inInputTerminal.12;


bRunningForward 	:= stDeviceMapping.inStatus.0;
bRunningReverse 	:= stDeviceMapping.inStatus.1;
bFault 				:= stDeviceMapping.inStatus.3;
bWarning 			:= stDeviceMapping.inStatus.7;
bRemoteEnabled		:= stDeviceMapping.inStatus.9;
bFrequencyMatching	:= stDeviceMapping.inStatus.12;
bConnectionError	:= stDeviceMapping.inStatus.15;
bECDisconnected		:= stDeviceMapping.ibWcState;

stDeviceMapping.onFrequencyRef 		:= REAL_TO_UINT(rFreq * 100.0);

bDriveOK := (eDeviceStatus>=4);
bError := eDeviceStatus < eOmronStatus.AWATING_RESET;
END_ACTION

ACTION aSetStatus:
IF bFault AND stDeviceMapping.inSTOActive THEN
	eDeviceStatus := eOmronStatus.AWATING_RESET;
ELSIF bFault THEN
	eDeviceStatus := eOmronStatus.FAULT;
ELSIF bECDisconnected THEN
	eDeviceStatus := eOmronStatus.DRIVE_DISCONNECTED;
ELSIF bConnectionError THEN
	eDeviceStatus := eOmronStatus.CONNECTION_ERROR;
ELSIF bWarning THEN
	eDeviceStatus := eOmronStatus.WARNING;
ELSIF (bRunningForward OR bRunningReverse) AND bFrequencyMatching THEN
	eDeviceStatus := eOmronStatus.RUNNING;
ELSIF bRemoteEnabled THEN
	eDeviceStatus := eOmronStatus.READY;

END_IF
END_ACTION

METHOD PROTECTED CreateEvents
VAR_INPUT
END_VAR
// Add your event creation here
F_CreateAllEventsInClass(Alarms		:= MotionLinxAlarms,
						 ClassSize	:= SIZEOF(TC_EVENTS.MotionlinxAI_Axis),
						 pInitEvent := ADR(TC_EVENTS.MotionlinxAI_Axis.InitReferenceEvent),
						 Prefix		:= Name);

// Super call to base
SUPER^.CreateEvents();
END_METHOD

METHOD CyclicLogic
VAR_INPUT
END_VAR
IF NOT _InitComplete THEN
	_InitComplete := Initialize();
	RETURN;
END_IF

SUPER^.CyclicLogic();

//Read data from Parameters

aInputMapping();
aSetStatus();
END_METHOD

METHOD Disable : BOOL
VAR_INPUT
END_VAR
bEnabled := FALSE;
IF DriveState >= eDriveStates.STOPPED THEN
	RequestedState := eDriveStates.DISABLED;
END_IF
END_METHOD

PROPERTY Drive_State : eDriveStates
GET
Drive_State	:= DriveState;
END_GET
END_PROPERTY

METHOD Enable : BOOL
VAR_INPUT
END_VAR
bEnabled := TRUE;
bResetTried := FALSE;
IF DriveState >= eDriveStates.DISABLED THEN
	RequestedState := eDriveStates.STOPPED;
END_IF
END_METHOD

PROPERTY FaultLocation : STRING(50)
GET
FaultLocation := sDriveName;
END_GET
END_PROPERTY

PROPERTY HasFault : BOOL
GET
HasFault := DriveState = eDriveStates.FAULT;
END_GET
END_PROPERTY

METHOD PROTECTED HMICommunication
VAR_INPUT
END_VAR
SUPER^.HMICommunication();

//Handle the requests to extend and retract
IF ComponentBase_HMI.Status.HMIControlAvailable THEN
	IF MotionlinxAI_HMI.Command.Extend THEN
//		Extend();
	ELSIF MotionlinxAI_HMI.Command.Retract THEN
//		Retract();
	END_IF
END_IF

//Update HMI status info
//Cylinder_HMI.Status.Extended	:= _Extended;
//Cylinder_HMI.Status.Extending	:= _Extending;
//Cylinder_HMI.Status.Retracted	:= _Retracted;
//Cylinder_HMI.Status.Retracting	:= _Retracting;
//Cylinder_HMI.Config.ExtendTime	:= _ExtendTime;
//Cylinder_HMI.Config.RetractTime := _RetractTime;
END_METHOD

PROPERTY IsReady : BOOL
GET
IsReady := DriveState >= eDriveStates.DISABLED;
END_GET
END_PROPERTY

PROPERTY IsRunning : BOOL
GET
IsRunning := bFrequencyMatching;
END_GET
END_PROPERTY

METHOD PROTECTED Monitoring
VAR_INPUT
END_VAR
_Busy	 := IsRunning;
_Error	 := eDeviceStatus < eOmronStatus.AWATING_RESET;
_ErrorID := ;//eError;
SUPER^.Monitoring();
END_METHOD

PROPERTY STO_Active : bool
GET
END_GET
END_PROPERTY

END_FUNCTION_BLOCK

// ---- Machine/Components/Drives/Omron/Old System/DM_Omron/DM_Omron_Drive.TcPOU
FUNCTION_BLOCK DM_Omron_Drive IMPLEMENTS iDM_DriveHealth
VAR CONSTANT
	MIN_LIBRARY_VERSION : DM_LIBRARY_VERSION := DM_LIBRARY_VERSION.V_20240925;
END_VAR
VAR_INPUT
	bRun : BOOL;
	rFreq : REAL;
	bReverse: BOOL := FALSE;
	nAccelTime : UINT := 200;
	nDecelTime : UINT := 200;	
END_VAR
VAR_IN_OUT
	stDeviceMapping : stOmronDriveMapping;
END_VAR
VAR_OUTPUT
	DriveState : eDriveStates := eDriveStates.FAULT;
	
	bDI1: BOOL;
	bDI2: BOOL;
	bDI3: BOOL;
	bDI4: BOOL;
	bDI5: BOOL;
	bDI6: BOOL;
	bDI7: BOOL;
	bEN1: BOOL;
	bEN2: BOOL;
	bDriveOK : BOOL;
	sOmronDriveStatus: STRING;			
	
END_VAR
VAR
	RequestedState : eDriveStates := eDriveStates.AWAITING_RESET;	

	bEnabled : BOOL;
	bInitReversed : BOOL;
	bError : BOOL;
	
	
	eDeviceStatus : eOmronStatus;
	
	bRunningForward : BOOL;
	bRunningReverse : BOOL;
	bFault : BOOL;
	bWarning : BOOL;
	bRemoteEnabled : BOOL;
	bFrequencyMatching : BOOL;
	bConnectionError : BOOL;
	bECDisconnected : BOOL;
	
	blinkErrorAck : FB_BLINKER_PLAY;
	
	tpErrorReset : TP;
	bResetReq : BOOL;
	
	sDriveName : STRING(50);
	tonFailedStartTimeout : TON;
	bResetTried: BOOL;
END_VAR

//Set Drive Status
aSetStatus();
aStateMachine();
aInputMapping();

stDeviceMapping.onDecelTime := nDecelTime;
stDeviceMapping.onAccelTime := nAccelTime;

//Run Stop Control
IF DriveState >= eDriveStates.STOPPED THEN
	IF bRun THEN
	 	RequestedState := eDriveStates.RUNNING;
	ELSE
		RequestedState := eDriveStates.STOPPED;
	END_IF
END_IF


IF DriveState >= eDriveStates.STARTING THEN
	IF bReverse XOR bInitReversed THEN
		stDeviceMapping.onCommand.0 := FALSE;
		stDeviceMapping.onCommand.1 := TRUE;
	ELSE
		stDeviceMapping.onCommand.0 := TRUE;
		stDeviceMapping.onCommand.1 := FALSE;
	END_IF
ELSE	
	stDeviceMapping.onCommand.0 := stDeviceMapping.onCommand.1 := FALSE;
END_IF

tonFailedStartTimeout(IN:= DriveState = eDriveStates.RUNNING AND stDeviceMapping.inMotorCurrent = 0 , PT := T#5S);
IF tonFailedStartTimeout.Q THEN 
	IF NOT bResetTried THEN 
		Reset();
		bResetTried := TRUE;
	ELSE
		Disable();
	END_IF
END_IF

ACTION aInputMapping:
bDI1 := stDeviceMapping.inInputTerminal.2;
bDI2 := stDeviceMapping.inInputTerminal.3;
bDI3 := stDeviceMapping.inInputTerminal.4;
bDI4 := stDeviceMapping.inInputTerminal.5;
bDI5 := stDeviceMapping.inInputTerminal.6;
bDI6 := stDeviceMapping.inInputTerminal.0; 
bDI7 := stDeviceMapping.inInputTerminal.1;
bEN1 := stDeviceMapping.inInputTerminal.11;
bEN2 := stDeviceMapping.inInputTerminal.12;


bRunningForward 	:= stDeviceMapping.inStatus.0;
bRunningReverse 	:= stDeviceMapping.inStatus.1;
bFault 				:= stDeviceMapping.inStatus.3;
bWarning 			:= stDeviceMapping.inStatus.7;
bRemoteEnabled		:= stDeviceMapping.inStatus.9;
bFrequencyMatching	:= stDeviceMapping.inStatus.12;
bConnectionError	:= stDeviceMapping.inStatus.15;
bECDisconnected		:= stDeviceMapping.ibWcState;

stDeviceMapping.onFrequencyRef 		:= REAL_TO_UINT(rFreq * 100.0);

bDriveOK := (eDeviceStatus>=4);
bError := eDeviceStatus < eOmronStatus.AWATING_RESET;
END_ACTION

ACTION aSetStatus:
IF bFault AND stDeviceMapping.inSTOActive THEN
	eDeviceStatus := eOmronStatus.AWATING_RESET;
ELSIF bFault THEN
	eDeviceStatus := eOmronStatus.FAULT;
ELSIF bECDisconnected THEN
	eDeviceStatus := eOmronStatus.DRIVE_DISCONNECTED;
ELSIF bConnectionError THEN
	eDeviceStatus := eOmronStatus.CONNECTION_ERROR;
ELSIF bWarning THEN
	eDeviceStatus := eOmronStatus.WARNING;
ELSIF (bRunningForward OR bRunningReverse) AND bFrequencyMatching THEN
	eDeviceStatus := eOmronStatus.RUNNING;
ELSIF bRemoteEnabled THEN
	eDeviceStatus := eOmronStatus.READY;

END_IF
END_ACTION

ACTION aStateMachine:
CASE DriveState OF
	////////////////////////////////////////////////////
	eDriveStates.FAULT:
	
		blinkErrorAck(bStartPulser := bError, tTimeDelayON := T#0.1S, tTimeDelayOFF := T#0.1S, tTimeGap := T#0.5S, nNoOfBlinks := 3, bPulseComplete => stDeviceMapping.onCommand.7);
		IF NOT bError THEN
			DriveState := eDriveStates.AWAITING_RESET;
		END_IF;
		
	////////////////////////////////////////////////////
	eDriveStates.FAULT_STOPPING:
		Disable();
		DriveState := eDriveStates.FAULT;
		
	////////////////////////////////////////////////////
	eDriveStates.AWAITING_RESET:
		IF RequestedState = eDriveStates.RESET THEN
			DriveState := eDriveStates.RESET;
		END_IF;
		IF berror THEN			
			DriveState := eDriveStates.FAULT;
		END_IF
	
	////////////////////////////////////////////////////
	eDriveStates.RESET:	
		IF NOT bError AND bRemoteEnabled THEN
			DriveState := RequestedState := eDriveStates.STOPPED;
		END_IF
		IF berror THEN			
			DriveState := eDriveStates.FAULT;
		END_IF
	
	////////////////////////////////////////////////////
	eDriveStates.DISABLED:		
		IF bEnabled THEN
			DriveState := eDriveStates.STOPPED;
		END_IF;
		IF berror THEN			
			DriveState := eDriveStates.FAULT;
		END_IF
					
	////////////////////////////////////////////////////	
	eDriveStates.STOPPED:
		IF RequestedState = eDriveStates.RUNNING THEN
			DriveState := eDriveStates.RUNNING;
		END_IF
		
		IF RequestedState = eDriveStates.RESET THEN
			DriveState := eDriveStates.AWAITING_RESET;
		END_IF
		
		IF NOT bEnabled OR RequestedState = eDriveStates.DISABLED THEN
			DriveState := eDriveStates.DISABLED;
		END_IF
		IF bError THEN			
			DriveState := eDriveStates.FAULT;
		END_IF

	////////////////////////////////////////////////////		
	eDriveStates.STOPPING:
		IF stDeviceMapping.inOutputFrequency = 0 OR bError THEN
			DriveState := eDriveStates.STOPPED;
		END_IF
	
	////////////////////////////////////////////////////	
	eDriveStates.STARTING:
		IF bFrequencyMatching THEN
			DriveState := eDriveStates.RUNNING;
		END_IF
		
		IF bError OR RequestedState < eDriveStates.STARTING THEN
			DriveState := eDriveStates.STOPPING;
		END_IF
		
	////////////////////////////////////////////////////
	eDriveStates.RUNNING:		
		IF RequestedState <> eDriveStates.RUNNING OR NOT bRun OR bError THEN
			DriveState := eDriveStates.STOPPING;
		END_IF
		
END_CASE
END_ACTION

METHOD Disable : BOOL
VAR_INPUT
END_VAR
bEnabled := FALSE;
IF DriveState >= eDriveStates.STOPPED THEN
	RequestedState := eDriveStates.DISABLED;
END_IF
END_METHOD

METHOD Enable : BOOL
VAR_INPUT
END_VAR
bEnabled := TRUE;
bResetTried := FALSE;
IF DriveState >= eDriveStates.DISABLED THEN
	RequestedState := eDriveStates.STOPPED;
END_IF
END_METHOD

PROPERTY FaultLocation : STRING(50)
GET
FaultLocation := sDriveName;
END_GET
END_PROPERTY

METHOD FB_init : BOOL
VAR_INPUT
	bInitRetains : BOOL; // if TRUE, the retain variables are initialized (warm start / cold start)
	bInCopyCode : BOOL;  // if TRUE, the instance afterwards gets moved into the copy code (online change)
	bReversed : BOOL;
	sName : STRING(50);
END_VAR
bInitReversed := bReversed;
sDriveName := sName;
END_METHOD

PROPERTY HasFault : BOOL
GET
HasFault := DriveState = eDriveStates.FAULT;
END_GET
END_PROPERTY

PROPERTY IsReady : BOOL
GET
IsReady := DriveState >= eDriveStates.DISABLED;
END_GET
END_PROPERTY

PROPERTY IsRunning : BOOL
GET
IsRunning := bFrequencyMatching;
END_GET
END_PROPERTY

PROPERTY Name : STRING(50)
GET
Name:=sDriveName;
END_GET
SET
sDriveName:=Name;
END_SET
END_PROPERTY

METHOD Reset : BOOL
VAR_INPUT
END_VAR
RequestedState := eDriveStates.RESET;
END_METHOD

END_FUNCTION_BLOCK

// ---- Machine/Components/Drives/Roller Drives/2 Motor Drive/Axis/FB_Drive_Type_1_Axis.TcPOU
(*	This FB is used for a single output solenoid 
	It uses the times to say when Extended/Retracted  	
	It starts assuming retracted and the output off.
*)
FUNCTION_BLOCK FB_Drive_Type_1_Axis EXTENDS FB_ComponentBase IMPLEMENTS I_Drive_Type_1_Axis
VAR
	//Output
	Input AT %I* : BOOL;
	Output AT %Q* : BOOL;

	// Internal variables
	_ExtendRequest	: BOOL;
	_RetractRequest : BOOL;
	_Extended		: BOOL;
	_Retracted		: BOOL;
	_Extending		: BOOL;
	_Retracting		: BOOL;
	_ExtendTime		: LREAL := 1000; // Default time 1s
	_RetractTime	: LREAL := 1000; // Default time 1s

	// Timer for Extend/Retract
	Extend_TON	  : TON;
	Retract_TON	  : TON;
	Extend_RTRIG  : R_TRIG;
	Retract_RTRIG : R_TRIG;
	Counter	:INT;

	//HMI 
	Cylinder_HMI : ST_Cylinder_HMI;
END_VAR

METHOD PROTECTED CreateEvents
VAR_INPUT
END_VAR
SUPER^.CreateEvents();
END_METHOD

METHOD CyclicLogic
Counter	:= Counter + 1;

//One shot the requests
Extend_RTRIG(CLK := _ExtendRequest);
Retract_RTRIG(CLK := _RetractRequest);

//Handle Extend
IF Extend_RTRIG.Q THEN
	Output			:= TRUE;
	_Extending		:= TRUE;
	_Retracting		:= FALSE;
	_Retracted		:= FALSE;
	_RetractRequest := FALSE;
END_IF

//Handle Retract
IF Retract_RTRIG.Q THEN
	Output		   := FALSE;
	_Extending	   := FALSE;
	_Retracting	   := TRUE;
	_Extended	   := FALSE;
	_ExtendRequest := FALSE;
END_IF

//Handle the time to Extend/Retract
Extend_TON(IN := _Extending, PT := LREAL_TO_TIME(_ExtendTime));
Retract_TON(IN := _Retracting, PT := LREAL_TO_TIME(_RetractTime));
IF Extend_TON.Q THEN
	_Extended  := TRUE;
	_Extending := FALSE;
END_IF

IF Retract_TON.Q THEN
	_Retracted	:= TRUE;
	_Retracting := FALSE;
END_IF

SUPER^.CyclicLogic();
END_METHOD

METHOD Drive : BOOL
VAR_INPUT
END_VAR
END_METHOD

METHOD PROTECTED HMICommunication
VAR_INPUT
END_VAR
SUPER^.HMICommunication();

//Handle the requests to extend and retract
IF ComponentBase_HMI.Status.HMIControlAvailable THEN
	IF Cylinder_HMI.Command.Extend THEN
//		Extend();
	ELSIF Cylinder_HMI.Command.Retract THEN
//		Retract();
	END_IF
END_IF

//Update HMI status info
Cylinder_HMI.Status.Extended	:= _Extended;
Cylinder_HMI.Status.Extending	:= _Extending;
Cylinder_HMI.Status.Retracted	:= _Retracted;
Cylinder_HMI.Status.Retracting	:= _Retracting;
Cylinder_HMI.Config.ExtendTime	:= _ExtendTime;
Cylinder_HMI.Config.RetractTime := _RetractTime;
END_METHOD

//! @summary Basic component initialization logic
METHOD PROTECTED Initialize : BOOL;

//! @description This method is called by <c>CyclicLogic()</c> as required
//Set the cylinder to retracted
IF Output THEN
	_Extended  := TRUE;
	_Retracted := FALSE;
ELSE
	_Extended  := FALSE;
	_Retracted := TRUE;
END_IF

_Extending		:= FALSE;
_ExtendRequest	:= FALSE;
_Retracting		:= FALSE;
_RetractRequest := FALSE;

//Call base class Initialize
Initialize := SUPER^.Initialize();
END_METHOD

METHOD PROTECTED Monitoring
VAR_INPUT
END_VAR
_Busy	 := _Extending OR _Retracting;
_Error	 := FALSE;
_ErrorID := 0;
SUPER^.Monitoring();
END_METHOD

PROPERTY Position : real
GET
END_GET
SET
END_SET
END_PROPERTY

END_FUNCTION_BLOCK

// ---- Machine/Components/Drives/Roller Drives/2 Motor Drive/FB_Drive_Type_1_Controller.TcPOU
(*	This FB is used for a single output solenoid 
	It uses the times to say when Extended/Retracted  	
	It starts assuming retracted and the output off.
*)
FUNCTION_BLOCK FB_Drive_Type_1_Controller EXTENDS FB_ComponentBase
VAR
	//Output
	Drive_1_Left	:FB_Drive_Type_1_Axis	;	//Reference to Drive FB for Motor 1/Left
	Drive_2_Right	:FB_Drive_Type_1_Axis	;
	//Drive_2_Right	ref to:FB_Drive_Type_1_Axis ; 	Reference to Drive FB for Motor 1/Left

	// Internal variables
	_ExtendRequest	: BOOL;
	_RetractRequest : BOOL;
	_Extended		: BOOL;
	_Retracted		: BOOL;
	_Extending		: BOOL;
	_Retracting		: BOOL;
	_ExtendTime		: LREAL := 1000; // Default time 1s
	_RetractTime	: LREAL := 1000; // Default time 1s

	// Timer for Extend/Retract
	Extend_TON	  : TON;
	Retract_TON	  : TON;
	Extend_RTRIG  : R_TRIG;
	Retract_RTRIG : R_TRIG;

	//HMI 
	Cylinder_HMI : ST_Cylinder_HMI;
END_VAR

METHOD PROTECTED CreateEvents
VAR_INPUT
END_VAR
SUPER^.CreateEvents();
END_METHOD

METHOD CyclicLogic
Drive_1_Left.CyclicLogic();
Drive_2_Right.CyclicLogic();


//One shot the requests
Extend_RTRIG(CLK := _ExtendRequest);
Retract_RTRIG(CLK := _RetractRequest);

//Handle Extend
//IF Extend_RTRIG.Q THEN
//	Output			:= TRUE;
//	_Extending		:= TRUE;
//	_Retracting		:= FALSE;
//	_Retracted		:= FALSE;
//	_RetractRequest := FALSE;
//END_IF

////Handle Retract
//IF Retract_RTRIG.Q THEN
//	Output		   := FALSE;
//	_Extending	   := FALSE;
//	_Retracting	   := TRUE;
//	_Extended	   := FALSE;
//	_ExtendRequest := FALSE;
//END_IF

////Handle the time to Extend/Retract
//Extend_TON(IN := _Extending, PT := LREAL_TO_TIME(_ExtendTime));
//Retract_TON(IN := _Retracting, PT := LREAL_TO_TIME(_RetractTime));
//IF Extend_TON.Q THEN
//	_Extended  := TRUE;
//	_Extending := FALSE;
//END_IF

//IF Retract_TON.Q THEN
//	_Retracted	:= TRUE;
//	_Retracting := FALSE;
//END_IF

SUPER^.CyclicLogic();
END_METHOD

METHOD PROTECTED HMICommunication
VAR_INPUT
END_VAR
SUPER^.HMICommunication();

//Handle the requests to extend and retract
IF ComponentBase_HMI.Status.HMIControlAvailable THEN
	IF Cylinder_HMI.Command.Extend THEN
//		Extend();
	ELSIF Cylinder_HMI.Command.Retract THEN
//		Retract();
	END_IF
END_IF

//Update HMI status info
Cylinder_HMI.Status.Extended	:= _Extended;
Cylinder_HMI.Status.Extending	:= _Extending;
Cylinder_HMI.Status.Retracted	:= _Retracted;
Cylinder_HMI.Status.Retracting	:= _Retracting;
Cylinder_HMI.Config.ExtendTime	:= _ExtendTime;
Cylinder_HMI.Config.RetractTime := _RetractTime;
END_METHOD

//! @summary Basic component initialization logic
METHOD PROTECTED Initialize : BOOL;

//! @description This method is called by <c>CyclicLogic()</c> as required
//Set the cylinder to retracted
//IF Output THEN
//	_Extended  := TRUE;
//	_Retracted := FALSE;
//ELSE
//	_Extended  := FALSE;
//	_Retracted := TRUE;
//END_IF

_Extending		:= FALSE;
_ExtendRequest	:= FALSE;
_Retracting		:= FALSE;
_RetractRequest := FALSE;

//Call base class Initialize
Initialize := SUPER^.Initialize();
END_METHOD

METHOD PROTECTED Monitoring
VAR_INPUT
END_VAR
_Busy	 := _Extending OR _Retracting;
_Error	 := FALSE;
_ErrorID := 0;
SUPER^.Monitoring();
END_METHOD

END_FUNCTION_BLOCK

// ---- Machine/Components/Relay/Relay_Pulse.TcPOU
FUNCTION_BLOCK Relay_Pulse IMPLEMENTS I_Relay
VAR
	output AT %Q* : BOOL;
	bFirstRun	:BOOL :=true;	//Only ran for 1 cycle
	rt_ON	:r_trig;
	rt_OFF	:r_trig;
	_SwitchOn		:BOOL;
	_SwitchOff	:BOOL;
	tp_Pulse	:TP;
	_tPulseTime	:TIME:=T#500MS;
	_Invert_Output	:BOOL;
	ft_Output	:f_trig;
	_ON	:BOOL;
	_OFF	:BOOL;
END_VAR

METHOD Cyclic
VAR_INPUT
END_VAR

tp_Pulse(in:=_SwitchOn OR _SwitchOff, pt:=_tPulseTime(*, Q => output*));
//ft_Output (CLK:= output);
IF _Invert_Output THEN
	output	:= NOT tp_Pulse.Q;
	ft_Output (CLK:= NOT output);
ELSE
	output	:= tp_Pulse.Q;
	ft_Output (CLK:= output);
END_IF

IF ft_Output.Q THEN
	_SwitchOn		:=FALSE;
	_SwitchOff	:=FALSE;
	rt_ON(CLK:=FALSE);
	rt_OFF(CLK:=FALSE);
	
END_IF

IF _Invert_Output THEN
	IF _SwitchOn AND NOT output THEN
		_ON		:= TRUE;
		_Off	:=FALSE;
	ELSIF 
		_SwitchOff AND NOT output THEN
		_ON		:= FALSE;
		_Off	:=TRUE;
	END_IF
ELSE
	IF _SwitchOn AND output THEN
		_ON		:= TRUE;
		_Off	:=FALSE;
	ELSIF 
		_SwitchOff AND output THEN
		_ON		:= FALSE;
		_Off	:=TRUE;
	END_IF
END_IF



(*IF _Invert_Output THEN
	IF _SwitchOn AND NOT output THEN
		_ON		:= FALSE;
		_Off	:=TRUE;
	ELSIF 
		_SwitchOff AND NOT output THEN
		_ON		:= TRUE;
		_Off	:=FALSE;
	END_IF
ELSE
	IF _SwitchOn AND output THEN
		_ON		:= TRUE;
		_Off	:=FALSE;
	ELSIF 
		_SwitchOff AND output THEN
		_ON		:= FALSE;
		_Off	:=TRUE;
	END_IF
END_IF*)
END_METHOD

METHOD FB_init : BOOL
VAR_INPUT
	bInitRetains : BOOL; // if TRUE, the retain variables are initialized (warm start / cold start)
	bInCopyCode : BOOL;  // if TRUE, the instance afterwards gets moved into the copy code (online change)
	Invert_Output	:BOOL;
END_VAR
_Invert_Output	:= Invert_Output;
IF  bFirstRun THEN 
	IF _Invert_Output THEN
		output	:=TRUE;
	END_IF
	_OFF	:= TRUE;
	bFirstRun	:= FALSE;
END_IF
//_Plusled_Output	:=Plusled_Output;
END_METHOD

{attribute 'monitoring' := 'variable'}
PROPERTY OFF : BOOL
GET
OFF	:= _OFF;
END_GET
END_PROPERTY

PROPERTY ON : Bool
GET
ON := _ON;
END_GET
END_PROPERTY

METHOD PUBLIC SwitchOff
VAR_INPUT
END_VAR
rt_OFF(CLK:= TRUE);
IF rt_OFF.Q THEN
	_SwitchOff	:=TRUE;
END_IF
END_METHOD

METHOD PUBLIC SwitchOn
VAR_INPUT
END_VAR
rt_ON(CLK:= TRUE);
IF rt_ON.Q THEN
	_SwitchOn	:=TRUE;
END_IF
END_METHOD

PROPERTY tPulseTime : Time
SET
_tPulseTime	:= tPulseTime;
END_SET
END_PROPERTY

END_FUNCTION_BLOCK

// ---- Machine/Components/Vision/Cognex/FB_A100.TcPOU
(*	This FB is used for a single output solenoid 
	It uses the times to say when Extended/Retracted  	
	It starts assuming retracted and the output off.
*)
FUNCTION_BLOCK FB_A100 EXTENDS FB_ComponentBase IMPLEMENTS I_Cylinder
VAR
	//Output
	Output AT %Q* : BOOL;

	// Internal variables
	_ExtendRequest	: BOOL;
	_RetractRequest : BOOL;
	_Extended		: BOOL;
	_Retracted		: BOOL;
	_Extending		: BOOL;
	_Retracting		: BOOL;
	_ExtendTime		: LREAL := 1000; // Default time 1s
	_RetractTime	: LREAL := 1000; // Default time 1s

	// Timer for Extend/Retract
	Extend_TON	  : TON;
	Retract_TON	  : TON;
	Extend_RTRIG  : R_TRIG;
	Retract_RTRIG : R_TRIG;

	//HMI 
	Cylinder_HMI : ST_Cylinder_HMI;
END_VAR

METHOD PROTECTED CreateEvents
VAR_INPUT
END_VAR
SUPER^.CreateEvents();
END_METHOD

METHOD CyclicLogic
//One shot the requests
Extend_RTRIG(CLK := _ExtendRequest);
Retract_RTRIG(CLK := _RetractRequest);

//Handle Extend
IF Extend_RTRIG.Q THEN
	Output			:= TRUE;
	_Extending		:= TRUE;
	_Retracting		:= FALSE;
	_Retracted		:= FALSE;
	_RetractRequest := FALSE;
END_IF

//Handle Retract
IF Retract_RTRIG.Q THEN
	Output		   := FALSE;
	_Extending	   := FALSE;
	_Retracting	   := TRUE;
	_Extended	   := FALSE;
	_ExtendRequest := FALSE;
END_IF

//Handle the time to Extend/Retract
Extend_TON(IN := _Extending, PT := LREAL_TO_TIME(_ExtendTime));
Retract_TON(IN := _Retracting, PT := LREAL_TO_TIME(_RetractTime));
IF Extend_TON.Q THEN
	_Extended  := TRUE;
	_Extending := FALSE;
END_IF

IF Retract_TON.Q THEN
	_Retracted	:= TRUE;
	_Retracting := FALSE;
END_IF

SUPER^.CyclicLogic();
END_METHOD

METHOD Extend
_ExtendRequest	:= TRUE;
_RetractRequest := FALSE;
END_METHOD

PROPERTY Extended : BOOL
GET
Extended := _Extended;
END_GET
END_PROPERTY

PROPERTY ExtendTime : LREAL
GET
ExtendTime := _ExtendTime;
END_GET
SET
END_SET
END_PROPERTY

METHOD PROTECTED HMICommunication
VAR_INPUT
END_VAR
SUPER^.HMICommunication();

//Handle the requests to extend and retract
IF ComponentBase_HMI.Status.HMIControlAvailable THEN
	IF Cylinder_HMI.Command.Extend THEN
		Extend();
	ELSIF Cylinder_HMI.Command.Retract THEN
		Retract();
	END_IF
END_IF

//Update HMI status info
Cylinder_HMI.Status.Extended	:= _Extended;
Cylinder_HMI.Status.Extending	:= _Extending;
Cylinder_HMI.Status.Retracted	:= _Retracted;
Cylinder_HMI.Status.Retracting	:= _Retracting;
Cylinder_HMI.Config.ExtendTime	:= _ExtendTime;
Cylinder_HMI.Config.RetractTime := _RetractTime;
END_METHOD

//! @summary Basic component initialization logic
METHOD PROTECTED Initialize : BOOL;

//! @description This method is called by <c>CyclicLogic()</c> as required
//Set the cylinder to retracted
IF Output THEN
	_Extended  := TRUE;
	_Retracted := FALSE;
ELSE
	_Extended  := FALSE;
	_Retracted := TRUE;
END_IF

_Extending		:= FALSE;
_ExtendRequest	:= FALSE;
_Retracting		:= FALSE;
_RetractRequest := FALSE;

//Call base class Initialize
Initialize := SUPER^.Initialize();
END_METHOD

METHOD PROTECTED Monitoring
VAR_INPUT
END_VAR
_Busy	 := _Extending OR _Retracting;
_Error	 := FALSE;
_ErrorID := 0;
SUPER^.Monitoring();
END_METHOD

METHOD Retract
_ExtendRequest	:= FALSE;
_RetractRequest := TRUE;
END_METHOD

PROPERTY Retracted : BOOL
GET
Retracted := _Retracted;
END_GET
END_PROPERTY

PROPERTY RetractTime : LREAL
GET
RetractTime := _RetractTime;
END_GET
SET
_RetractTime := RetractTime;
END_SET
END_PROPERTY

END_FUNCTION_BLOCK

// ---- Machine/EquipmentModules/Conveyors/FB_Robot_Outfeed_Conveyor_Module.TcPOU
FUNCTION_BLOCK FB_Robot_Outfeed_Conveyor_Module EXTENDS FB_Station_Module
VAR
END_VAR

(*
Controls the outfeed conveyor for a robot, when item in place, indicates to robot to run object removal and allows another object to be fed in




*)

METHOD PROTECTED FINAL Execute
VAR_INPUT
END_VAR
CASE _CurrentMode OF
	//=================================PRODUCTION MODE==================================
	E_PMLUnitMode.ePMLUnitMode_Production:
		CASE SequenceState OF
			0:
				NoStateTasksToComplete := FALSE;
				IF 	Sensor.Active THEN
					SequenceState := SequenceState + 10;
				END_IF
		
			10:
			//	NoStateTasksToComplete := FALSE;
			
				Deceleration := Recipe.Axis.Deceleration;
				Axis.Stop();
				SequenceState := SequenceState + 10;

			20:
				IF Axis.Stopped THEN
					SequenceState := SequenceState + 10;
				END_IF

			30:
				StateComplete();
		END_CASE
	
	i	:= i +1;
	
		(* Run the sequence to make products 
		 Unwind Runs Slowly 
		 Pull Wheels Run 
		 Jaws Seal, and Repeat until production reached*)
//		sealTrig(CLK := SequenceState = 10);
//		IF sealTrig.Q THEN
//			partTimeStart := F_GetActualDcTime64();
//			sealTimeStart := partTimeStart;
//		END_IF

//		pulltrig(CLK := SequenceState = 20);
//		IF pulltrig.Q THEN
//			pullTimeStart := F_GetActualDcTime64();
//		END_IF

	//	Buffer_1.ChangeState(E_PMLCommand.ePMLCommand_Start);

		
		
//		IF THIS^.Sealer.sealbar.InTempRange THEN
//			CASE SequenceState OF
//				0: //Started
//					Unwind.ChangeState(E_PMLCommand.ePMLCommand_Start);
//					IF Unwind.CurrentState = E_PMLState.ePMLState_Execute THEN
//						SequenceState := SequenceState + 10;
//					END_IF

//				10: // SEAL First
//					Sealer.ChangeState(E_PMLCommand.ePMLCommand_Start);
//					IF Sealer.CurrentState = E_PMLState.ePMLState_Complete THEN
//						Sealer.ChangeState(E_PMLCommand.ePMLCommand_Reset);
//						SequenceState := SequenceState + 10;
//						SealTimeEnd	  := F_GetActualDcTime64();
//						sealingTime	  := ULINT_TO_LREAL(sealtimeEnd - sealTimeStart) * 1E-9;
//					END_IF

//				20: // Run Pullwheels
//					PullWheels.ChangeState(E_PMLCommand.ePMLCommand_Start);
//					IF PullWheels.CurrentState = E_PMLState.ePMLState_Complete THEN
//						partTimeEnd	  := F_GetActualDcTime64();
//						parts		  := parts + 1;
//						SequenceState := 10;
//						PullWheels.ChangeState(E_PMLCommand.ePMLCommand_Reset);
//						pullTimeEnd := F_GetActualDcTime64();
//						pullingTime := ULINT_TO_LREAL(pullTimeEnd - pullTimeStart) * 1E-9;
//					END_IF
//			END_CASE
//		ELSE
//			ChangeState(E_PMLCommand.ePMLCommand_Suspend);
//		END_IF

	//=================================MAINTENANCE MODE==================================	
	E_PMLUnitMode.ePMLUnitMode_Maintenance:
		;

	//=================================MANUAL MODE==================================
	E_PMLUnitMode.ePMLUnitMode_Manual:
		;
END_CASE
END_METHOD

END_FUNCTION_BLOCK

// ---- Machine/EquipmentModules/Conveyors/FB_SingleDrive_Conveyor_With_Out_Sensor.TcPOU
FUNCTION_BLOCK FB_SingleDrive_Conveyor_With_Out_Sensor EXTENDS FB_PackML_BaseModule
VAR
	// Sub module definitions here

	// List of sub modules
	ipSubModules_Init : ARRAY[1..Parameters_PackML_Base.MAX_NO_OF_SUBMODULES] OF I_PackML_BaseModule := [];

	// Component definitions here
//	Axis   : FB_Component_BasicAxis := (Name := 'Axis');
//	Sensor : FB_DigitalSensor		:= (Name := 'Sensor');
	Previous_Sensor	:I_DigitalSensorBase;
	OutFeed_Sensor	:I_DigitalSensorBase;

	//Alarms for this module
	ConveyorModuleAlarms : ARRAY[1..CONVEYOR_MODULE_ALARM_COUNT] OF FB_TcAlarm;

	//Data for recipe
	Recipe : ST_Closer_Recipe;

	(*Parameters from PackTags for module
    //_Param  : ARRAY[1..10] OF ST_Descriptor2;*)
	_Report : ARRAY[1..10] OF ST_Descriptor2;

	//HMI Control for EM
	fbControlSourceHMI : FB_ControlSource_HMI;
END_VAR

VAR CONSTANT
	//reports 
	FAULT : INT := 1;

	//Alarms
	CONVEYOR_MODULE_ALARM_COUNT : INT := 5;
END_VAR

//Simulation variables for messaging
VAR
	ErrorInput : BOOL;
	WarnInput  : BOOL;
	InfoInput  : BOOL;
END_VAR

(*
Execute = Run conveyor
			if no infeed from previous for 1min go to idle - stop drive, wait for previous outfeed or previous operation busy? ?
			If out feed blocked, then stop at sensor - blocked until next is clear
			
			




*)

METHOD PROTECTED Aborting
VAR_INPUT
END_VAR
CASE SequenceState OF
	0:
		NoStateTasksToComplete := FALSE;
		SequenceState		   := SequenceState + 10;

	10:
	//	Axis.Stop();
	//	IF Axis.Stopped THEN
			SequenceState := SequenceState + 10;
	//	END_IF

	20:
		// Disable here
	//	Axis.Disable();

		// Check not enabled here
	//	IF NOT Axis.Enabled THEN
			SequenceState := SequenceState + 10;
	//	END_IF

	30:
		StateTasksComplete := TRUE;
END_CASE

SUPER^.Aborting();
END_METHOD

PROPERTY Acceleration : LREAL
SET
//Recipe.Axis.Acceleration := Acceleration;
END_SET
END_PROPERTY

METHOD PROTECTED Clearing
VAR_INPUT
END_VAR
CASE SequenceState OF
	0:
		NoStateTasksToComplete := FALSE;
		SequenceState		   := SequenceState + 10;

	10:
		//Reset any alarms that get latched
		ConveyorModuleAlarms[E_Unwind.StartTimeout].Clear(0, 0);
		SequenceState := SequenceState + 10;

	20:
		// Enable here
	//	Axis.Enable();

		// Check enabled here
	//	IF Axis.Enabled THEN
			SequenceState := SequenceState + 10;
	//	END_IF

	30:
		StateTasksComplete := TRUE;
END_CASE

SUPER^.Clearing();
END_METHOD

METHOD PROTECTED CreateEvents
VAR_INPUT
END_VAR
// Add your event creation here
F_CreateAllEventsInClass(Alarms		:= ConveyorModuleAlarms,
						 ClassSize	:= SIZEOF(TC_EVENTS.Unwind),
						 pInitEvent := ADR(TC_EVENTS.Unwind.InitReferenceEvent),
						 Prefix		:= Name);

// Super call to base
SUPER^.CreateEvents();
END_METHOD

METHOD CyclicLogic
VAR_INPUT
END_VAR
IF NOT _InitComplete THEN
	_InitComplete := Initialize();
	RETURN;
END_IF

SUPER^.CyclicLogic();

//HMI control for EM
fbControlSourceHMI.CyclicLogic();

//Set the current alarm severity for this module
_CurrentAlarmSeverity := F_GetMaxSeverityRaised(Alarms := ConveyorModuleAlarms, CurrentSeverity := _CurrentAlarmSeverity);
IF _CurrentAlarmSeverity >= TcEventSeverity.Error THEN
	ChangeState(E_PMLCommand.ePMLCommand_Abort);
END_IF

//CyclicLogic_Simulation();
END_METHOD

METHOD CyclicLogic_Simulation
VAR_INPUT
END_VAR
(*	
This is just for testing. Real hardware can be setup in other places
Here the alarms will raise and clear on its own if the input changes	
*)

//Generic Alarms for Testing
IF ErrorInput AND NOT UnwindAlarms[E_Unwind.AlarmMessage].bRaised THEN
	RaiseAlarm2Args(UnwindAlarms[E_Unwind.AlarmMessage], '', '');
ELSIF NOT ErrorInput AND UnwindAlarms[E_Unwind.AlarmMessage].bRaised THEN
	UnwindAlarms[E_Unwind.AlarmMessage].Clear(0, 0);
END_IF

IF WarnInput AND NOT UnwindAlarms[E_Unwind.WarnMessage].bRaised THEN
	RaiseAlarm2Args(UnwindAlarms[E_Unwind.WarnMessage], '', '');
ELSIF NOT WarnInput AND UnwindAlarms[E_Unwind.WarnMessage].bRaised THEN
	UnwindAlarms[E_Unwind.WarnMessage].Clear(0, 0);
END_IF

IF InfoInput AND NOT UnwindAlarms[E_Unwind.InfoMessage].bRaised THEN
	RaiseAlarm2Args(UnwindAlarms[E_Unwind.InfoMessage], '', '');
ELSIF NOT InfoInput AND UnwindAlarms[E_Unwind.InfoMessage].bRaised THEN
	UnwindAlarms[E_Unwind.InfoMessage].Clear(0, 0);
END_IF
END_METHOD

METHOD FB_init : BOOL
VAR_INPUT
	bInitRetains : BOOL; // if TRUE, the retain variables are initialized (warm start / cold start)
	bInCopyCode : BOOL;  // if TRUE, the instance afterwards gets moved into the copy code (online change)
	OutFeed_Sensor	:I_DigitalSensorBase;
END_VAR
this^.	OutFeed_Sensor	:=OutFeed_Sensor;
END_METHOD

//! @summary Basic module initialization logic
METHOD PROTECTED Initialize : BOOL;
VAR
	i						 : UDINT;
	varInfo					 : __SYSTEM.VAR_INFO;
	AllSubUnitsInitialized	 : BOOL := TRUE;
	AllComponentsInitialized : BOOL := TRUE;
END_VAR

//! @description This method is called by <c>CyclicLogic()</c> as required
Initialize := FALSE;
CASE DescendantSequenceState OF
	0:
	//	RegisterComponent(Axis);
	//	RegisterComponent(Sensor);
		_LogModeChanges			:= FALSE;
		_LogStateChanges		:= FALSE;
		DescendantSequenceState := DescendantSequenceState + 10;

	10:
		//Setup Custom modes here

		(*CustomModes(eMode                          :=,
                    sName                          :=,
                    bDisableClearing               :=,
                    bDisableStarting               :=,
                    bDisableSuspended              :=,
                    bDisableStopping               :=,
                    bDisableAborting               :=,
                    bDisableHolding                :=,
                    bDisableHeld                   :=,
                    bDisableUnholding              :=,
                    bDisableSuspending             :=,
                    bDisableUnsuspending           :=,
                    bDisableResetting              :=,
                    bDisableIdle                   :=,
                    bDisableCompleting             :=,
                    bDisableComplete               :=,
                    bEnableUnitModeChangeStopped   :=,
                    bEnableUnitModeChangeIdle      :=,
                    bEnableUnitModeChangeSuspended :=,
                    bEnableUnitModeChangeExecute   :=,
                    bEnableUnitModeChangeAborted   :=,
                    bEnableUnitModeChangeHeld      :=,
                    bEnableUnitModeChangeComplete  :=,
                    bError                         =>,
                    nErrorId                       =>);*)
		DescendantSequenceState := DescendantSequenceState + 10;

	20:
		//Copy Mode names
		FOR i := 1 TO 3 DO
			ModeNames[i] := F_UnitModeToString(UDINT_TO_DINT(i));
		END_FOR

		Initialize_TagData();
		RegisterExternalController(Controller := fbControlSourceHMI);
		fbControlSourceHMI.CyclicLogic();

		//Set the Parent Response here
		_ParentFaultResponseDefinitions[TcEventSeverity.Error] := E_AlarmResponse.Hold_Immediate;
		DescendantSequenceState								   := DescendantSequenceState + 10;

	30:
		//Call the Super
		IF SUPER^.Initialize() THEN
			DescendantSequenceState := DescendantSequenceState + 10;
		END_IF

	40:
		Initialize := TRUE;
END_CASE
END_METHOD

METHOD Initialize_TagData
VAR_INPUT
END_VAR
//Recipe
//Recipe.Axis.Velocity	 := 100;
//Recipe.Axis.Acceleration := 1000;

//Report
_Report[FAULT].ID	:= TO_DINT(3 * 10 + 1);
_Report[FAULT].Name := 'Fault ID';
_Report[FAULT].Unit := 'n/a';
END_METHOD

METHOD RaiseAlarm2Args
VAR_IN_OUT
	Alarm : FB_TcAlarm; //Alarm to be raised
END_VAR

VAR_INPUT
	String_1 : STRING; //First String Parameter (The Name of this component will be applied first automatically)
	String_2 : STRING; //Second String Parameter
END_VAR
F_RaiseAlarmWithStringParameters(Alarm	  := Alarm,
								 String_1 := Name,
								 String_2 := String_1,
								 String_3 := String_2);
END_METHOD

METHOD PROTECTED Starting
VAR_INPUT
END_VAR

VAR_INST
	StartTimer : TON;
END_VAR
CASE _CurrentMode OF
	//=================================PRODUCTION MODE==================================
	E_PMLUnitMode.ePMLUnitMode_Production:
		CASE SequenceState OF
			0:
				// Delay 1 scan to make sure timer is off.  Not guarnteed from last time where it finished.
				NoStateTasksToComplete := FALSE;
				SequenceState		   := SequenceState + 10;

			10:
				NoStateTasksToComplete := FALSE;
//				Axis.Velocity		   := Recipe.LeftAxis;
//				Axis.Acceleration	   := Recipe.Axis.Acceleration;
//				Axis.MoveVelocity(Velocity := Recipe.Axis.Velocity, AbortPrevious := FALSE);
				SequenceState := SequenceState + 10;

			20:
			//	IF Axis.Busy THEN
					SequenceState := SequenceState + 10;
			//	END_IF

				IF StartTimer.Q AND NOT ConveyorModuleAlarms[E_Unwind.StartTimeout].bRaised THEN
					RaiseAlarm2Args(ConveyorModuleAlarms[E_Unwind.StartTimeout], '', '');
					SequenceState := SequenceState + 10;
				END_IF

			30:
				StateTasksComplete := TRUE;
		END_CASE

	//=================================MAINTENANCE & MANUAL MODE==================================
	E_PMLUnitMode.ePMLUnitMode_Maintenance, E_PMLUnitMode.ePMLUnitMode_Manual:
		;
END_CASE

SUPER^.Starting();
StartTimer(IN := (SequenceState = 10 OR SequenceState = 20), PT := T#3S);
END_METHOD

METHOD PROTECTED Stopping
VAR_INPUT
END_VAR
CASE _CurrentMode OF
	//=================================PRODUCTION MODE==================================
	E_PMLUnitMode.ePMLUnitMode_Production:
		CASE SequenceState OF
			0:
				NoStateTasksToComplete := FALSE;
			//	Axis.Stop();
				SequenceState := SequenceState + 10;

			10:
			//	IF Axis.Stopped THEN
					SequenceState := SequenceState + 10;
			//	END_IF

			20:
				StateTasksComplete := TRUE;
		END_CASE

	//=================================MAINTENANCE & MANUAL MODE==================================
	E_PMLUnitMode.ePMLUnitMode_Maintenance, E_PMLUnitMode.ePMLUnitMode_Manual:
		;
END_CASE

SUPER^.Stopping();
END_METHOD

PROPERTY Velocity : LREAL
SET
//Recipe.Axis.Velocity := Velocity;
END_SET
END_PROPERTY

END_FUNCTION_BLOCK

// ---- Machine/EquipmentModules/Conveyors/FB_SingleDrive_Conveyor_With_Out_Sensor_And_Stopper.TcPOU
FUNCTION_BLOCK FB_SingleDrive_Conveyor_With_Out_Sensor_And_Stopper EXTENDS FB_SingleDrive_Conveyor_With_Out_Sensor

VAR
END_VAR

END_FUNCTION_BLOCK

// ---- Machine/EquipmentModules/Conveyors/FB_Single_Drive_Outfeed_Sensor.TcPOU
FUNCTION_BLOCK FB_Single_Drive_Outfeed_Sensor EXTENDS FB_PackML_BaseModule
VAR
	//Axis Controller Status
	_Controller_Sts	:ST_Controller_Status ;

	// Sub module definitions here

	// List of sub modules
	ipSubModules_Init : ARRAY[1..Parameters_PackML_Base.MAX_NO_OF_SUBMODULES] OF I_PackML_BaseModule := [];

	// Component definitions here
//	Axis_Sensors   : FB_Component_BasicAxis := (Name := 'Axis');
	Axis   : FB_MotionlinxAI_Axis:=(Controller_Sts	:= _Controller_Sts);
	Sensor : FB_DigitalSensor		:= (Name := 'Sensor', DebounceMode := E_DebounceMode.SimpleFlickerFilter, DebounceTime := T#250MS, Inverted    := FALSE, SimulationInput:= FALSE, SimulationMode := E_SensorSimulationMode.InputDriven) ;


	//Alarms for this module
	ConveyorAlarms : ARRAY[1..CONVEYOR_ALARM_COUNT] OF FB_TcAlarm;

	//Data for recipe
	Recipe : ST_ConveyorRecipe;

	(*Parameters from PackTags for module
    //_Param  : ARRAY[1..10] OF ST_Descriptor2;*)
	_Report : ARRAY[1..10] OF ST_Descriptor2;

	//HMI Control for EM
	fbControlSourceHMI : FB_ControlSource_HMI;
	
	Enable_Drive	:BOOL;
	Disable_Drive	:BOOL;
	Emergency_Stop	:bool;
	Start_Drive		:BOOL;
	Stop_Drive		:BOOL;
END_VAR



VAR CONSTANT
	//reports 
	FAULT : INT := 1;

	//Alarms
	CONVEYOR_ALARM_COUNT : INT := 5;
END_VAR

//Simulation variables for messaging
VAR
	ErrorInput : BOOL;
	WarnInput  : BOOL;
	InfoInput  : BOOL;
END_VAR

METHOD PROTECTED Aborting
VAR_INPUT
END_VAR
CASE SequenceState OF
	0:
		NoStateTasksToComplete := FALSE;
		SequenceState		   := SequenceState + 10;

	10:
		Axis.Stop();
		IF Axis.Stopped THEN
			SequenceState := SequenceState + 10;
		END_IF

	20:
		// Disable here
		Axis.Disable();

		// Check not enabled here
		IF NOT Axis.Enabled THEN
			SequenceState := SequenceState + 10;
		END_IF

	30:
		StateTasksComplete := TRUE;
END_CASE

SUPER^.Aborting();
END_METHOD

PROPERTY Acceleration : int
SET
Recipe.Axis.Acceleration := Acceleration;
END_SET
END_PROPERTY

METHOD PROTECTED Clearing
VAR_INPUT
END_VAR
CASE SequenceState OF
	0:
		NoStateTasksToComplete := FALSE;
		SequenceState		   := SequenceState + 10;

	10:
		//Reset any alarms that get latched
		ConveyorAlarms[E_Unwind.StartTimeout].Clear(0, 0);
		SequenceState := SequenceState + 10;

	20:
		// Enable here
		Axis.Enable();

		// Check enabled here
		IF Axis.Enabled THEN
			SequenceState := SequenceState + 10;
		END_IF

	30:
		StateTasksComplete := TRUE;
END_CASE

SUPER^.Clearing();
END_METHOD

PROPERTY Controller_Sts : ST_Controller_Status
SET
_Controller_Sts	:=Controller_Sts;
END_SET
END_PROPERTY

METHOD PROTECTED CreateEvents
VAR_INPUT
END_VAR
// Add your event creation here
F_CreateAllEventsInClass(Alarms		:= ConveyorAlarms,
						 ClassSize	:= SIZEOF(TC_EVENTS.Unwind),
						 pInitEvent := ADR(TC_EVENTS.Unwind.InitReferenceEvent),
						 Prefix		:= Name);

// Super call to base
SUPER^.CreateEvents();
END_METHOD

METHOD CyclicLogic
VAR_INPUT
END_VAR
IF NOT _InitComplete THEN
	_InitComplete := Initialize();
	RETURN;
END_IF

SUPER^.CyclicLogic();

//Conveyor goes to idle and stop the conveyor if no input for 1 minute?
//Conveyor wont start if following conveyor in error or not running goes to blocked?


//HMI control for EM
fbControlSourceHMI.CyclicLogic();

//Set the current alarm severity for this module
_CurrentAlarmSeverity := F_GetMaxSeverityRaised(Alarms := ConveyorAlarms, CurrentSeverity := _CurrentAlarmSeverity);
IF _CurrentAlarmSeverity >= TcEventSeverity.Error THEN
	ChangeState(E_PMLCommand.ePMLCommand_Abort);
END_IF

Axis.Controller_Sts	:= _Controller_Sts;

//Axis.Sensors;
//Axis.Controller_Sts:= iController_Sensors ;
//CyclicLogic_Simulation();

//Quick cotrol for testing

Recipe.Axis.MaxSpeed;
IF Emergency_Stop	 THEN
	Axis.EmergencyStop();
	Emergency_Stop	:= FALSE;
END_IF


IF Enable_Drive THEN
	Axis.Enable();
	Enable_Drive	:= FALSE;
END_IF


IF Disable_Drive THEN
	Axis.Disable();
	Disable_Drive	:= FALSE;
END_IF

IF Start_Drive THEN
	Axis.Acceleration := Recipe.Axis.Acceleration;
	Axis.Velocity := Recipe.Axis.Velocity;
	Axis.Start();
	IF not Axis.Stopped THEN
		Start_Drive	:= FALSE;
	END_IF
END_IF

IF Stop_Drive THEN
	Axis.Deceleration := Recipe.Axis.Deceleration;
//	Axis.Velocity := Recipe.Axis.Velocity;
	Axis.Stop();
	IF Axis.Stopped THEN
		Stop_Drive	:= FALSE;
	END_IF
END_IF
END_METHOD

METHOD CyclicLogic_Simulation
VAR_INPUT
END_VAR
(*	
This is just for testing. Real hardware can be setup in other places
Here the alarms will raise and clear on its own if the input changes	
*)

//Generic Alarms for Testing
IF ErrorInput AND NOT UnwindAlarms[E_Unwind.AlarmMessage].bRaised THEN
	RaiseAlarm2Args(UnwindAlarms[E_Unwind.AlarmMessage], '', '');
ELSIF NOT ErrorInput AND UnwindAlarms[E_Unwind.AlarmMessage].bRaised THEN
	UnwindAlarms[E_Unwind.AlarmMessage].Clear(0, 0);
END_IF

IF WarnInput AND NOT UnwindAlarms[E_Unwind.WarnMessage].bRaised THEN
	RaiseAlarm2Args(UnwindAlarms[E_Unwind.WarnMessage], '', '');
ELSIF NOT WarnInput AND UnwindAlarms[E_Unwind.WarnMessage].bRaised THEN
	UnwindAlarms[E_Unwind.WarnMessage].Clear(0, 0);
END_IF

IF InfoInput AND NOT UnwindAlarms[E_Unwind.InfoMessage].bRaised THEN
	RaiseAlarm2Args(UnwindAlarms[E_Unwind.InfoMessage], '', '');
ELSIF NOT InfoInput AND UnwindAlarms[E_Unwind.InfoMessage].bRaised THEN
	UnwindAlarms[E_Unwind.InfoMessage].Clear(0, 0);
END_IF
END_METHOD

PROPERTY Deceleration : int
SET
Recipe.Axis.Deceleration := Deceleration;
END_SET
END_PROPERTY

//! @summary Basic module initialization logic
METHOD PROTECTED Initialize : BOOL;
VAR
	i						 : UDINT;
	varInfo					 : __SYSTEM.VAR_INFO;
	AllSubUnitsInitialized	 : BOOL := TRUE;
	AllComponentsInitialized : BOOL := TRUE;
END_VAR

//! @description This method is called by <c>CyclicLogic()</c> as required
	Axis.MaxSpeed := Recipe.Axis.MaxSpeed;

//https://beckhoff-usa-community.github.io/SPT-Libraries/Getting_Started/PackML%20Overview.html
Initialize := FALSE;
CASE DescendantSequenceState OF
	0:
		RegisterComponent(Axis);
		RegisterComponent(Sensor);
		_LogModeChanges			:= FALSE;
		_LogStateChanges		:= FALSE;
		DescendantSequenceState := DescendantSequenceState + 10;

	10:
		//Setup Custom modes here

		CustomModes(eMode                          :=,
                    sName                          :=,
                    bDisableClearing               :=true,		// Is there a sequence that has to happen in clearing or can I sit in Stopped and perform the clear?
                    bDisableStarting               :=,
                    bDisableSuspended              :=false,	//Upstream or downstream are blocked
                    bDisableStopping               :=,
                    bDisableAborting               :=false,		//Ramp down the drives needed?
                    bDisableHolding                :=false,		//Nothing for operator to do ie refil
                    bDisableHeld                   :=false,		//Nothing for operator to do ie refil
                    bDisableUnholding              :=false,		//Nothing for operator to do ie refil
                    bDisableSuspending             :=false,	//Upstream or downstream are blocked
                    bDisableUnsuspending           :=false,	//Upstream or downstream are blocked
                    bDisableResetting              :=,
                    bDisableIdle                   :=,
                    bDisableCompleting             :=TRUE,	//Disable of coneyor or 1 part only the conveyor
                    bDisableComplete               :=true,
                    bEnableUnitModeChangeStopped   :=,
                    bEnableUnitModeChangeIdle      :=,
                    bEnableUnitModeChangeSuspended :=,
                    bEnableUnitModeChangeExecute   :=,
                    bEnableUnitModeChangeAborted   :=,
                    bEnableUnitModeChangeHeld      :=,
                    bEnableUnitModeChangeComplete  :=,
                    bError                         =>,
                    nErrorId                       =>);
		DescendantSequenceState := DescendantSequenceState + 10;

	20:
		//Copy Mode names
		FOR i := 1 TO 3 DO
			ModeNames[i] := F_UnitModeToString(UDINT_TO_DINT(i));
		END_FOR

		Initialize_TagData();
		RegisterExternalController(Controller := fbControlSourceHMI);
		fbControlSourceHMI.CyclicLogic();

		//Set the Parent Response here
		_ParentFaultResponseDefinitions[TcEventSeverity.Error] := E_AlarmResponse.Hold_Immediate;
		DescendantSequenceState								   := DescendantSequenceState + 10;

	30:
		//Call the Super
		IF SUPER^.Initialize() THEN
			DescendantSequenceState := DescendantSequenceState + 10;
		END_IF

	40:
		Initialize := TRUE;
END_CASE
END_METHOD

METHOD Initialize_TagData
VAR_INPUT
END_VAR
//Recipe
Recipe.Axis.Velocity	 := 50;
Recipe.Axis.Acceleration := 1000;
Recipe.Axis.Deceleration := 500;
Recipe.Axis.MaxSpeed	 := 100;

//Report
_Report[FAULT].ID	:= TO_DINT(3 * 10 + 1);
_Report[FAULT].Name := 'Fault ID';
_Report[FAULT].Unit := 'n/a';
END_METHOD

METHOD RaiseAlarm2Args
VAR_IN_OUT
	Alarm : FB_TcAlarm; //Alarm to be raised
END_VAR

VAR_INPUT
	String_1 : STRING; //First String Parameter (The Name of this component will be applied first automatically)
	String_2 : STRING; //Second String Parameter
END_VAR
F_RaiseAlarmWithStringParameters(Alarm	  := Alarm,
								 String_1 := Name,
								 String_2 := String_1,
								 String_3 := String_2);
END_METHOD

METHOD PROTECTED Starting
VAR_INPUT
END_VAR

VAR_INST
	StartTimer : TON;
END_VAR
CASE _CurrentMode OF
	//=================================PRODUCTION MODE==================================
	E_PMLUnitMode.ePMLUnitMode_Production:
		CASE SequenceState OF
			0:
				// Delay 1 scan to make sure timer is off.  Not guarnteed from last time where it finished.
				NoStateTasksToComplete := FALSE;
				SequenceState		   := SequenceState + 10;

			10:
				NoStateTasksToComplete := FALSE;
		
				
				Axis.Velocity		   := Recipe.Axis.Velocity;
				Axis.Acceleration	   := Recipe.Axis.Acceleration;
				Axis.Start();
		//		Axis.MoveVelocity(Velocity := Recipe.Axis.Velocity, AbortPrevious := FALSE);
				SequenceState := SequenceState + 10;

			20:
				IF Axis.Busy THEN
					SequenceState := SequenceState + 10;
				END_IF

				IF StartTimer.Q AND NOT ConveyorAlarms[E_Unwind.StartTimeout].bRaised THEN
					RaiseAlarm2Args(ConveyorAlarms[E_Unwind.StartTimeout], '', '');
					SequenceState := SequenceState + 10;
				END_IF

			30:
				StateTasksComplete := TRUE;
		END_CASE

	//=================================MAINTENANCE & MANUAL MODE==================================
	E_PMLUnitMode.ePMLUnitMode_Maintenance, E_PMLUnitMode.ePMLUnitMode_Manual:
		;
END_CASE

SUPER^.Starting();
StartTimer(IN := (SequenceState = 10 OR SequenceState = 20), PT := T#3S);
END_METHOD

METHOD PROTECTED Stopping
VAR_INPUT
END_VAR
CASE _CurrentMode OF
	//=================================PRODUCTION MODE==================================
	E_PMLUnitMode.ePMLUnitMode_Production:
		CASE SequenceState OF
			0:
				NoStateTasksToComplete := FALSE;
			//	Axis.Stop();
				Deceleration := Recipe.Axis.Deceleration;
				Axis.Stop();
				SequenceState := SequenceState + 10;

			10:
				IF Axis.Stopped THEN
					SequenceState := SequenceState + 10;
				END_IF

			20:
				StateTasksComplete := TRUE;
		END_CASE

	//=================================MAINTENANCE & MANUAL MODE==================================
	E_PMLUnitMode.ePMLUnitMode_Maintenance, E_PMLUnitMode.ePMLUnitMode_Manual:
		;
END_CASE

SUPER^.Stopping();
END_METHOD

PROPERTY Velocity : int
SET
Recipe.Axis.Velocity := Velocity;
END_SET
END_PROPERTY

END_FUNCTION_BLOCK

// ---- Machine/EquipmentModules/FB_Diverter_Module.TcPOU
FUNCTION_BLOCK FB_Diverter_Module EXTENDS FB_PackML_BaseModule
VAR
	// Sub module definitions here

	// List of sub modules
	ipSubModules_Init : ARRAY[1..Parameters_PackML_Base.MAX_NO_OF_SUBMODULES] OF I_PackML_BaseModule := [];

	// Component definitions here
//	Axis   : FB_Component_BasicAxis := (Name := 'Axis');
	Drive_1	:I_Drive_Type_1_Axis;
	Drive_2	:I_Drive_Type_1_Axis;
	Sensor : FB_DigitalSensor		:= (Name := 'Sensor');

	//Alarms for this module
	DiverterAlarms : ARRAY[1..DIVERTER_ALARM_COUNT] OF FB_TcAlarm;

	//Data for recipe
	Recipe : ST_DiverterRecipe;

	(*Parameters from PackTags for module
    //_Param  : ARRAY[1..10] OF ST_Descriptor2;*)
	_Report : ARRAY[1..10] OF ST_Descriptor2;

	//HMI Control for EM
	fbControlSourceHMI : FB_ControlSource_HMI;
END_VAR

VAR CONSTANT
	//reports 
	FAULT : INT := 1;

	//Alarms
	DIVERTER_ALARM_COUNT : INT := 5;
END_VAR

//Simulation variables for messaging
VAR
	ErrorInput : BOOL;
	WarnInput  : BOOL;
	InfoInput  : BOOL;
END_VAR

METHOD PROTECTED Aborting
VAR_INPUT
END_VAR
CASE SequenceState OF
	0:
		NoStateTasksToComplete := FALSE;
		SequenceState		   := SequenceState + 10;

	10:
	//	Axis.Stop();
	//	IF Axis.Stopped THEN
			SequenceState := SequenceState + 10;
	//	END_IF

	20:
		// Disable here
	//	Axis.Disable();

		// Check not enabled here
	//	IF NOT Axis.Enabled THEN
			SequenceState := SequenceState + 10;
	//	END_IF

	30:
		StateTasksComplete := TRUE;
END_CASE

SUPER^.Aborting();
END_METHOD

PROPERTY Acceleration : LREAL
SET
//Recipe.Axis.Acceleration := Acceleration;
END_SET
END_PROPERTY

METHOD PROTECTED Clearing
VAR_INPUT
END_VAR
CASE SequenceState OF
	0:
		NoStateTasksToComplete := FALSE;
		SequenceState		   := SequenceState + 10;

	10:
		//Reset any alarms that get latched
		DiverterAlarms[E_Unwind.StartTimeout].Clear(0, 0);
		SequenceState := SequenceState + 10;

	20:
		// Enable here
	//	Axis.Enable();

		// Check enabled here
	//	IF Axis.Enabled THEN
			SequenceState := SequenceState + 10;
	//	END_IF

	30:
		StateTasksComplete := TRUE;
END_CASE

SUPER^.Clearing();
END_METHOD

METHOD PROTECTED CreateEvents
VAR_INPUT
END_VAR
// Add your event creation here
F_CreateAllEventsInClass(Alarms		:= DiverterAlarms,
						 ClassSize	:= SIZEOF(TC_EVENTS.Unwind),
						 pInitEvent := ADR(TC_EVENTS.Unwind.InitReferenceEvent),
						 Prefix		:= Name);

// Super call to base
SUPER^.CreateEvents();
END_METHOD

METHOD CyclicLogic
VAR_INPUT
END_VAR
IF NOT _InitComplete THEN
	_InitComplete := Initialize();
	RETURN;
END_IF

SUPER^.CyclicLogic();

//HMI control for EM
fbControlSourceHMI.CyclicLogic();

//Set the current alarm severity for this module
_CurrentAlarmSeverity := F_GetMaxSeverityRaised(Alarms := DiverterAlarms, CurrentSeverity := _CurrentAlarmSeverity);
IF _CurrentAlarmSeverity >= TcEventSeverity.Error THEN
	ChangeState(E_PMLCommand.ePMLCommand_Abort);
END_IF

//CyclicLogic_Simulation();
END_METHOD

METHOD CyclicLogic_Simulation
VAR_INPUT
END_VAR
(*	
This is just for testing. Real hardware can be setup in other places
Here the alarms will raise and clear on its own if the input changes	
*)

//Generic Alarms for Testing
IF ErrorInput AND NOT UnwindAlarms[E_Unwind.AlarmMessage].bRaised THEN
	RaiseAlarm2Args(UnwindAlarms[E_Unwind.AlarmMessage], '', '');
ELSIF NOT ErrorInput AND UnwindAlarms[E_Unwind.AlarmMessage].bRaised THEN
	UnwindAlarms[E_Unwind.AlarmMessage].Clear(0, 0);
END_IF

IF WarnInput AND NOT UnwindAlarms[E_Unwind.WarnMessage].bRaised THEN
	RaiseAlarm2Args(UnwindAlarms[E_Unwind.WarnMessage], '', '');
ELSIF NOT WarnInput AND UnwindAlarms[E_Unwind.WarnMessage].bRaised THEN
	UnwindAlarms[E_Unwind.WarnMessage].Clear(0, 0);
END_IF

IF InfoInput AND NOT UnwindAlarms[E_Unwind.InfoMessage].bRaised THEN
	RaiseAlarm2Args(UnwindAlarms[E_Unwind.InfoMessage], '', '');
ELSIF NOT InfoInput AND UnwindAlarms[E_Unwind.InfoMessage].bRaised THEN
	UnwindAlarms[E_Unwind.InfoMessage].Clear(0, 0);
END_IF
END_METHOD

METHOD FB_init : BOOL
VAR_INPUT
	bInitRetains : BOOL; // if TRUE, the retain variables are initialized (warm start / cold start)
	bInCopyCode : BOOL;  // if TRUE, the instance afterwards gets moved into the copy code (online change)
	Drive_1	:I_Drive_Type_1_Axis;
	Drive_2	:I_Drive_Type_1_Axis;
END_VAR
THIS^.Drive_1	:=	Drive_1 ;
THIS^.Drive_2	:=	Drive_2 ;
END_METHOD

//! @summary Basic module initialization logic
METHOD PROTECTED Initialize : BOOL;
VAR
	i						 : UDINT;
	varInfo					 : __SYSTEM.VAR_INFO;
	AllSubUnitsInitialized	 : BOOL := TRUE;
	AllComponentsInitialized : BOOL := TRUE;
END_VAR

//! @description This method is called by <c>CyclicLogic()</c> as required
Initialize := FALSE;
CASE DescendantSequenceState OF
	0:
	//	RegisterComponent(Axis);
	//	RegisterComponent(Drive_1);
		RegisterComponent(Sensor);
		_LogModeChanges			:= FALSE;
		_LogStateChanges		:= FALSE;
		DescendantSequenceState := DescendantSequenceState + 10;

	10:
		//Setup Custom modes here

		(*CustomModes(eMode                          :=,
                    sName                          :=,
                    bDisableClearing               :=,
                    bDisableStarting               :=,
                    bDisableSuspended              :=,
                    bDisableStopping               :=,
                    bDisableAborting               :=,
                    bDisableHolding                :=,
                    bDisableHeld                   :=,
                    bDisableUnholding              :=,
                    bDisableSuspending             :=,
                    bDisableUnsuspending           :=,
                    bDisableResetting              :=,
                    bDisableIdle                   :=,
                    bDisableCompleting             :=,
                    bDisableComplete               :=,
                    bEnableUnitModeChangeStopped   :=,
                    bEnableUnitModeChangeIdle      :=,
                    bEnableUnitModeChangeSuspended :=,
                    bEnableUnitModeChangeExecute   :=,
                    bEnableUnitModeChangeAborted   :=,
                    bEnableUnitModeChangeHeld      :=,
                    bEnableUnitModeChangeComplete  :=,
                    bError                         =>,
                    nErrorId                       =>);*)
		DescendantSequenceState := DescendantSequenceState + 10;

	20:
		//Copy Mode names
		FOR i := 1 TO 3 DO
			ModeNames[i] := F_UnitModeToString(UDINT_TO_DINT(i));
		END_FOR

		Initialize_TagData();
		RegisterExternalController(Controller := fbControlSourceHMI);
		fbControlSourceHMI.CyclicLogic();

		//Set the Parent Response here
		_ParentFaultResponseDefinitions[TcEventSeverity.Error] := E_AlarmResponse.Hold_Immediate;
		DescendantSequenceState								   := DescendantSequenceState + 10;

	30:
		//Call the Super
		IF SUPER^.Initialize() THEN
			DescendantSequenceState := DescendantSequenceState + 10;
		END_IF

	40:
		Initialize := TRUE;
END_CASE
END_METHOD

METHOD Initialize_TagData
VAR_INPUT
END_VAR
//Recipe
//Recipe.Axis.Velocity	 := 100;
//Recipe.Axis.Acceleration := 1000;

//Report
_Report[FAULT].ID	:= TO_DINT(3 * 10 + 1);
_Report[FAULT].Name := 'Fault ID';
_Report[FAULT].Unit := 'n/a';
END_METHOD

METHOD RaiseAlarm2Args
VAR_IN_OUT
	Alarm : FB_TcAlarm; //Alarm to be raised
END_VAR

VAR_INPUT
	String_1 : STRING; //First String Parameter (The Name of this component will be applied first automatically)
	String_2 : STRING; //Second String Parameter
END_VAR
F_RaiseAlarmWithStringParameters(Alarm	  := Alarm,
								 String_1 := Name,
								 String_2 := String_1,
								 String_3 := String_2);
END_METHOD

METHOD PROTECTED Starting
VAR_INPUT
END_VAR

VAR_INST
	StartTimer : TON;
END_VAR
CASE _CurrentMode OF
	//=================================PRODUCTION MODE==================================
	E_PMLUnitMode.ePMLUnitMode_Production:
		CASE SequenceState OF
			0:
				// Delay 1 scan to make sure timer is off.  Not guarnteed from last time where it finished.
				NoStateTasksToComplete := FALSE;
				SequenceState		   := SequenceState + 10;

			10:
				NoStateTasksToComplete := FALSE;
//				Axis.Velocity		   := Recipe.Axis.Velocity;
//				Axis.Acceleration	   := Recipe.Axis.Acceleration;
//				Axis.MoveVelocity(Velocity := Recipe.Axis.Velocity, AbortPrevious := FALSE);
				SequenceState := SequenceState + 10;

			20:
		//		IF Axis.Busy THEN
					SequenceState := SequenceState + 10;
		//		END_IF

				IF StartTimer.Q AND NOT DiverterAlarms[E_Unwind.StartTimeout].bRaised THEN
					RaiseAlarm2Args(DiverterAlarms[E_Unwind.StartTimeout], '', '');
					SequenceState := SequenceState + 10;
				END_IF

			30:
				StateTasksComplete := TRUE;
		END_CASE

	//=================================MAINTENANCE & MANUAL MODE==================================
	E_PMLUnitMode.ePMLUnitMode_Maintenance, E_PMLUnitMode.ePMLUnitMode_Manual:
		;
END_CASE

SUPER^.Starting();
StartTimer(IN := (SequenceState = 10 OR SequenceState = 20), PT := T#3S);
END_METHOD

METHOD PROTECTED Stopping
VAR_INPUT
END_VAR
CASE _CurrentMode OF
	//=================================PRODUCTION MODE==================================
	E_PMLUnitMode.ePMLUnitMode_Production:
		CASE SequenceState OF
			0:
				NoStateTasksToComplete := FALSE;
		//		Axis.Stop();
				SequenceState := SequenceState + 10;

			10:
		//		IF Axis.Stopped THEN
					SequenceState := SequenceState + 10;
		//		END_IF

			20:
				StateTasksComplete := TRUE;
		END_CASE

	//=================================MAINTENANCE & MANUAL MODE==================================
	E_PMLUnitMode.ePMLUnitMode_Maintenance, E_PMLUnitMode.ePMLUnitMode_Manual:
		;
END_CASE

SUPER^.Stopping();
END_METHOD

PROPERTY Velocity : LREAL
SET
//Recipe.Axis.Velocity := Velocity;
END_SET
END_PROPERTY

END_FUNCTION_BLOCK

// ---- Machine/EquipmentModules/FB_Labeler_Module.TcPOU
FUNCTION_BLOCK FB_Labeler_Module EXTENDS FB_PackML_BaseModule
VAR
	// Sub module definitions here
	Infeed_Vision_Sensor		: FB_Vision_Barcode_SubModule		:= (Name := 'Infeed_Vision_Sensor', LogStateChanges := TRUE);
	Labeler						: FB_Labeler_SubModule				:= (Name := 'Labeler', LogStateChanges := TRUE);
	Outfeed_Vision_Sensor		: FB_Vision_Barcode_SubModule		:= (Name := 'Outfeed_Vision_Sensor', LogStateChanges := TRUE);
	
	// List of sub modules
	ipSubModules_Init : ARRAY[1..Parameters_PackML_Base.MAX_NO_OF_SUBMODULES] OF I_PackML_BaseModule := [];

	// Component definitions here
//	Axis   : FB_Component_BasicAxis := (Name := 'Axis');
	Sensor : FB_DigitalSensor		:= (Name := 'Sensor');

	//Alarms for this module
	LabelerAlarms : ARRAY[1..LABELER_ALARM_COUNT] OF FB_TcAlarm;

	//Data for recipe
	Recipe : ST_LabelerRecipe;

	(*Parameters from PackTags for module
    //_Param  : ARRAY[1..10] OF ST_Descriptor2;*)
	_Report : ARRAY[1..10] OF ST_Descriptor2;

	//HMI Control for EM
	fbControlSourceHMI : FB_ControlSource_HMI;
END_VAR

VAR CONSTANT
	//reports 
	FAULT : INT := 1;

	//Alarms
	LABELER_ALARM_COUNT : INT := 5;
END_VAR

//Simulation variables for messaging
VAR
	ErrorInput : BOOL;
	WarnInput  : BOOL;
	InfoInput  : BOOL;
END_VAR

METHOD PROTECTED Aborting
VAR_INPUT
END_VAR
CASE SequenceState OF
	0:
		NoStateTasksToComplete := FALSE;
		SequenceState		   := SequenceState + 10;

	10:
	//	Axis.Stop();
	//	IF Axis.Stopped THEN
			SequenceState := SequenceState + 10;
	//	END_IF

	20:
		// Disable here
	//	Axis.Disable();

		// Check not enabled here
	//	IF NOT Axis.Enabled THEN
			SequenceState := SequenceState + 10;
	//	END_IF

	30:
		StateTasksComplete := TRUE;
END_CASE

SUPER^.Aborting();
END_METHOD

PROPERTY Acceleration : LREAL
SET
//Recipe.Axis.Acceleration := Acceleration;
END_SET
END_PROPERTY

METHOD PROTECTED Clearing
VAR_INPUT
END_VAR
CASE SequenceState OF
	0:
		NoStateTasksToComplete := FALSE;
		SequenceState		   := SequenceState + 10;

	10:
		//Reset any alarms that get latched
		LabelerAlarms[E_Unwind.StartTimeout].Clear(0, 0);
		SequenceState := SequenceState + 10;

	20:
		// Enable here
	//	Axis.Enable();

		// Check enabled here
	//	IF Axis.Enabled THEN
			SequenceState := SequenceState + 10;
	//	END_IF

	30:
		StateTasksComplete := TRUE;
END_CASE

SUPER^.Clearing();
END_METHOD

METHOD PROTECTED CreateEvents
VAR_INPUT
END_VAR
// Add your event creation here
F_CreateAllEventsInClass(Alarms		:= LabelerAlarms,
						 ClassSize	:= SIZEOF(TC_EVENTS.Unwind),
						 pInitEvent := ADR(TC_EVENTS.Unwind.InitReferenceEvent),
						 Prefix		:= Name);

// Super call to base
SUPER^.CreateEvents();
END_METHOD

METHOD CyclicLogic
VAR_INPUT
END_VAR
IF NOT _InitComplete THEN
	_InitComplete := Initialize();
	RETURN;
END_IF

SUPER^.CyclicLogic();

//HMI control for EM
fbControlSourceHMI.CyclicLogic();

//Set the current alarm severity for this module
_CurrentAlarmSeverity := F_GetMaxSeverityRaised(Alarms := LabelerAlarms, CurrentSeverity := _CurrentAlarmSeverity);
IF _CurrentAlarmSeverity >= TcEventSeverity.Error THEN
	ChangeState(E_PMLCommand.ePMLCommand_Abort);
END_IF

//CyclicLogic_Simulation();
END_METHOD

METHOD CyclicLogic_Simulation
VAR_INPUT
END_VAR
(*	
This is just for testing. Real hardware can be setup in other places
Here the alarms will raise and clear on its own if the input changes	
*)

//Generic Alarms for Testing
IF ErrorInput AND NOT UnwindAlarms[E_Unwind.AlarmMessage].bRaised THEN
	RaiseAlarm2Args(UnwindAlarms[E_Unwind.AlarmMessage], '', '');
ELSIF NOT ErrorInput AND UnwindAlarms[E_Unwind.AlarmMessage].bRaised THEN
	UnwindAlarms[E_Unwind.AlarmMessage].Clear(0, 0);
END_IF

IF WarnInput AND NOT UnwindAlarms[E_Unwind.WarnMessage].bRaised THEN
	RaiseAlarm2Args(UnwindAlarms[E_Unwind.WarnMessage], '', '');
ELSIF NOT WarnInput AND UnwindAlarms[E_Unwind.WarnMessage].bRaised THEN
	UnwindAlarms[E_Unwind.WarnMessage].Clear(0, 0);
END_IF

IF InfoInput AND NOT UnwindAlarms[E_Unwind.InfoMessage].bRaised THEN
	RaiseAlarm2Args(UnwindAlarms[E_Unwind.InfoMessage], '', '');
ELSIF NOT InfoInput AND UnwindAlarms[E_Unwind.InfoMessage].bRaised THEN
	UnwindAlarms[E_Unwind.InfoMessage].Clear(0, 0);
END_IF
END_METHOD

//! @summary Basic module initialization logic
METHOD PROTECTED Initialize : BOOL;
VAR
	i						 : UDINT;
	varInfo					 : __SYSTEM.VAR_INFO;
	AllSubUnitsInitialized	 : BOOL := TRUE;
	AllComponentsInitialized : BOOL := TRUE;
END_VAR

//! @description This method is called by <c>CyclicLogic()</c> as required
Initialize := FALSE;
CASE DescendantSequenceState OF
	0:
		RegisterSubModule(Infeed_Vision_Sensor);
		RegisterSubModule(Labeler);
		RegisterSubModule(Outfeed_Vision_Sensor);
		RegisterComponent(Sensor);
		_LogModeChanges			:= FALSE;
		_LogStateChanges		:= FALSE;
		DescendantSequenceState := DescendantSequenceState + 10;

	10:
		//Setup Custom modes here

		(*CustomModes(eMode                          :=,
                    sName                          :=,
                    bDisableClearing               :=,
                    bDisableStarting               :=,
                    bDisableSuspended              :=,
                    bDisableStopping               :=,
                    bDisableAborting               :=,
                    bDisableHolding                :=,
                    bDisableHeld                   :=,
                    bDisableUnholding              :=,
                    bDisableSuspending             :=,
                    bDisableUnsuspending           :=,
                    bDisableResetting              :=,
                    bDisableIdle                   :=,
                    bDisableCompleting             :=,
                    bDisableComplete               :=,
                    bEnableUnitModeChangeStopped   :=,
                    bEnableUnitModeChangeIdle      :=,
                    bEnableUnitModeChangeSuspended :=,
                    bEnableUnitModeChangeExecute   :=,
                    bEnableUnitModeChangeAborted   :=,
                    bEnableUnitModeChangeHeld      :=,
                    bEnableUnitModeChangeComplete  :=,
                    bError                         =>,
                    nErrorId                       =>);*)
		DescendantSequenceState := DescendantSequenceState + 10;

	20:
		//Copy Mode names
		FOR i := 1 TO 3 DO
			ModeNames[i] := F_UnitModeToString(UDINT_TO_DINT(i));
		END_FOR

		Initialize_TagData();
		RegisterExternalController(Controller := fbControlSourceHMI);
		fbControlSourceHMI.CyclicLogic();

		//Set the Parent Response here
		_ParentFaultResponseDefinitions[TcEventSeverity.Error] := E_AlarmResponse.Hold_Immediate;
		DescendantSequenceState								   := DescendantSequenceState + 10;

	30:
		//Call the Super
		IF SUPER^.Initialize() THEN
			DescendantSequenceState := DescendantSequenceState + 10;
		END_IF

	40:
		Initialize := TRUE;
END_CASE
END_METHOD

METHOD Initialize_TagData
VAR_INPUT
END_VAR
//Recipe
//Recipe.Axis.Velocity	 := 100;
//Recipe.Axis.Acceleration := 1000;

//Report
_Report[FAULT].ID	:= TO_DINT(3 * 10 + 1);
_Report[FAULT].Name := 'Fault ID';
_Report[FAULT].Unit := 'n/a';
END_METHOD

METHOD RaiseAlarm2Args
VAR_IN_OUT
	Alarm : FB_TcAlarm; //Alarm to be raised
END_VAR

VAR_INPUT
	String_1 : STRING; //First String Parameter (The Name of this component will be applied first automatically)
	String_2 : STRING; //Second String Parameter
END_VAR
F_RaiseAlarmWithStringParameters(Alarm	  := Alarm,
								 String_1 := Name,
								 String_2 := String_1,
								 String_3 := String_2);
END_METHOD

METHOD PROTECTED Starting
VAR_INPUT
END_VAR

VAR_INST
	StartTimer : TON;
END_VAR
CASE _CurrentMode OF
	//=================================PRODUCTION MODE==================================
	E_PMLUnitMode.ePMLUnitMode_Production:
		CASE SequenceState OF
			0:
				// Delay 1 scan to make sure timer is off.  Not guarnteed from last time where it finished.
				NoStateTasksToComplete := FALSE;
				SequenceState		   := SequenceState + 10;

			10:
				NoStateTasksToComplete := FALSE;
//				Axis.Velocity		   := Recipe.Axis.Velocity;
//				Axis.Acceleration	   := Recipe.Axis.Acceleration;
//				Axis.MoveVelocity(Velocity := Recipe.Axis.Velocity, AbortPrevious := FALSE);
				SequenceState := SequenceState + 10;

			20:
		//		IF Axis.Busy THEN
					SequenceState := SequenceState + 10;
		//		END_IF

				IF StartTimer.Q AND NOT LabelerAlarms[E_Unwind.StartTimeout].bRaised THEN
					RaiseAlarm2Args(LabelerAlarms[E_Unwind.StartTimeout], '', '');
					SequenceState := SequenceState + 10;
				END_IF

			30:
				StateTasksComplete := TRUE;
		END_CASE

	//=================================MAINTENANCE & MANUAL MODE==================================
	E_PMLUnitMode.ePMLUnitMode_Maintenance, E_PMLUnitMode.ePMLUnitMode_Manual:
		;
END_CASE

SUPER^.Starting();
StartTimer(IN := (SequenceState = 10 OR SequenceState = 20), PT := T#3S);
END_METHOD

METHOD PROTECTED Stopping
VAR_INPUT
END_VAR
CASE _CurrentMode OF
	//=================================PRODUCTION MODE==================================
	E_PMLUnitMode.ePMLUnitMode_Production:
		CASE SequenceState OF
			0:
				NoStateTasksToComplete := FALSE;
			//	Axis.Stop();
				SequenceState := SequenceState + 10;

			10:
			//	IF Axis.Stopped THEN
					SequenceState := SequenceState + 10;
			//	END_IF

			20:
				StateTasksComplete := TRUE;
		END_CASE

	//=================================MAINTENANCE & MANUAL MODE==================================
	E_PMLUnitMode.ePMLUnitMode_Maintenance, E_PMLUnitMode.ePMLUnitMode_Manual:
		;
END_CASE

SUPER^.Stopping();
END_METHOD

PROPERTY Velocity : LREAL
SET
//Recipe.Axis.Velocity := Velocity;
END_SET
END_PROPERTY

END_FUNCTION_BLOCK

// ---- Machine/EquipmentSubModules/FB_Vision_Barcode_SubModule.TcPOU
FUNCTION_BLOCK FB_Vision_Barcode_SubModule EXTENDS FB_PackML_BaseModule
VAR
	// Sub module definitions here

	// List of sub modules
	ipSubModules_Init : ARRAY[1..Parameters_PackML_Base.MAX_NO_OF_SUBMODULES] OF I_PackML_BaseModule := [];

	// Component definitions here
//	Axis   : FB_Component_BasicAxis := (Name := 'Axis');
	Sensor : FB_DigitalSensor		:= (Name := 'Sensor');

	//Alarms for this module
	VisionVolumeAlarms : ARRAY[1..VISION_VOLUME_ALARM_COUNT] OF FB_TcAlarm;

	//Data for recipe
	Recipe : ST_Vision_Volume_Recipe;

	(*Parameters from PackTags for module
    //_Param  : ARRAY[1..10] OF ST_Descriptor2;*)
	_Report : ARRAY[1..10] OF ST_Descriptor2;

	//HMI Control for EM
	fbControlSourceHMI : FB_ControlSource_HMI;
END_VAR

VAR CONSTANT
	//reports 
	FAULT : INT := 1;

	//Alarms
	VISION_VOLUME_ALARM_COUNT : INT := 5;
END_VAR

//Simulation variables for messaging
VAR
	ErrorInput : BOOL;
	WarnInput  : BOOL;
	InfoInput  : BOOL;
END_VAR

METHOD PROTECTED Aborting
VAR_INPUT
END_VAR
CASE SequenceState OF
	0:
		NoStateTasksToComplete := FALSE;
		SequenceState		   := SequenceState + 10;

	10:
	//	Axis.Stop();
	//	IF Axis.Stopped THEN
			SequenceState := SequenceState + 10;
	//	END_IF

	20:
		// Disable here
	//	Axis.Disable();

		// Check not enabled here
	//	IF NOT Axis.Enabled THEN
			SequenceState := SequenceState + 10;
	//	END_IF

	30:
		StateTasksComplete := TRUE;
END_CASE

SUPER^.Aborting();
END_METHOD

PROPERTY Acceleration : LREAL
SET
//Recipe.Axis.Acceleration := Acceleration;
END_SET
END_PROPERTY

METHOD PROTECTED Clearing
VAR_INPUT
END_VAR
CASE SequenceState OF
	0:
		NoStateTasksToComplete := FALSE;
		SequenceState		   := SequenceState + 10;

	10:
		//Reset any alarms that get latched
		VisionVolumeAlarms[E_Unwind.StartTimeout].Clear(0, 0);
		SequenceState := SequenceState + 10;

	20:
		// Enable here
	//	Axis.Enable();

		// Check enabled here
	//	IF Axis.Enabled THEN
			SequenceState := SequenceState + 10;
	//	END_IF

	30:
		StateTasksComplete := TRUE;
END_CASE

SUPER^.Clearing();
END_METHOD

METHOD PROTECTED CreateEvents
VAR_INPUT
END_VAR
// Add your event creation here
F_CreateAllEventsInClass(Alarms		:= VisionVolumeAlarms,
						 ClassSize	:= SIZEOF(TC_EVENTS.Unwind),
						 pInitEvent := ADR(TC_EVENTS.Unwind.InitReferenceEvent),
						 Prefix		:= Name);

// Super call to base
SUPER^.CreateEvents();
END_METHOD

METHOD CyclicLogic
VAR_INPUT
END_VAR
IF NOT _InitComplete THEN
	_InitComplete := Initialize();
	RETURN;
END_IF

SUPER^.CyclicLogic();

//HMI control for EM
fbControlSourceHMI.CyclicLogic();

//Set the current alarm severity for this module
_CurrentAlarmSeverity := F_GetMaxSeverityRaised(Alarms := VisionVolumeAlarms, CurrentSeverity := _CurrentAlarmSeverity);
IF _CurrentAlarmSeverity >= TcEventSeverity.Error THEN
	ChangeState(E_PMLCommand.ePMLCommand_Abort);
END_IF

//CyclicLogic_Simulation();
END_METHOD

METHOD CyclicLogic_Simulation
VAR_INPUT
END_VAR
(*	
This is just for testing. Real hardware can be setup in other places
Here the alarms will raise and clear on its own if the input changes	
*)

//Generic Alarms for Testing
IF ErrorInput AND NOT UnwindAlarms[E_Unwind.AlarmMessage].bRaised THEN
	RaiseAlarm2Args(UnwindAlarms[E_Unwind.AlarmMessage], '', '');
ELSIF NOT ErrorInput AND UnwindAlarms[E_Unwind.AlarmMessage].bRaised THEN
	UnwindAlarms[E_Unwind.AlarmMessage].Clear(0, 0);
END_IF

